(* POU LON/Module_1/Internal/FuSendCpValueReq_Module_1, ST *)
FUNCTION FuSendCpValueReq_Module_1 : BOOL
(******************************************)
(* Automatic generated code, do not edit! *)
(******************************************)
VAR_INPUT
	ptCp : POINTER TO BYTE;
	ptInternalUseOnly : POINTER TO BYTE;
	wCpIndex : WORD;
END_VAR
IF (ptCp <> 0) THEN
	IF ptInternalUseOnly^.0 = TRUE THEN
		OutDataTelegram_Module_1[0] := C2M_CP_VALUE_QRY;
		OutDataTelegram_Module_1[1] := WORD_TO_BYTE(wCpIndex AND 16#FF);
		OutDataTelegram_Module_1[2] := WORD_TO_BYTE((wCpIndex / 256) AND 16#FF);

		mbxModule_1.bTxPrio := 1;
		mbxModule_1.bTxProtID := 0;
		mbxModule_1.pbTxData := ADR(OutDataTelegram_Module_1);
		mbxModule_1.unTxLen := 3;
		mbxModule_1.MBX_SEND();

		IF (mbxModule_1.nError <> MBX_OK) THEN
			FuSendCpValueReq_Module_1 := FALSE;
			RETURN;
		END_IF
		ptInternalUseOnly^.0 := FALSE;
	END_IF
END_IF

FuSendCpValueReq_Module_1 := TRUE;
END_FUNCTION

(* POU LON/Shared/Internal/FuSnvtFilePosToRaw, ST *)
FUNCTION FuSnvtFilePosToRaw : BOOL
(******************************************)
(* Automatic generated code, do not edit! *)
(******************************************)
VAR_INPUT
	NvDataIn :  POINTER TO typSnvtFilePos;
	DataOut : POINTER TO ARRAY[0..5] OF BYTE;
END_VAR
VAR
END_VAR
DataOut^[0] := DINT_TO_BYTE(SHR(NvDataIn^.diRwPtr, 24));
DataOut^[1] := DINT_TO_BYTE(SHR(NvDataIn^.diRwPtr, 16));
DataOut^[2] := DINT_TO_BYTE(SHR(NvDataIn^.diRwPtr, 8));
DataOut^[3] := DINT_TO_BYTE(NvDataIn^.diRwPtr);

DataOut^[4] := WORD_TO_BYTE(SHR(NvDataIn^.wRwLength, 8));
DataOut^[5] := WORD_TO_BYTE(NvDataIn^.wRwLength);

FuSnvtFilePosToRaw := TRUE;
END_FUNCTION

(* POU LON/Shared/Internal/FuSnvtFileReqToRaw, ST *)
FUNCTION FuSnvtFileReqToRaw : BOOL
(******************************************)
(* Automatic generated code, do not edit! *)
(******************************************)
VAR_INPUT
	NvDataIn :  POINTER TO typSnvtFileReq;
	DataOut : POINTER TO ARRAY[0..11] OF BYTE;
END_VAR
VAR
END_VAR
DataOut^[0] := NvDataIn^.bRequest;

DataOut^[1] := WORD_TO_BYTE(SHR(NvDataIn^.wIndex, 8));
DataOut^[2] := WORD_TO_BYTE(NvDataIn^.wIndex);

DataOut^[3] := WORD_TO_BYTE(SHR(NvDataIn^.wReceiveTimeout, 8));
DataOut^[4] := WORD_TO_BYTE(NvDataIn^.wReceiveTimeout);

DataOut^[5] := NvDataIn^.abDestAddress[0];
DataOut^[6] := NvDataIn^.abDestAddress[1];
DataOut^[7] := NvDataIn^.abDestAddress[2];
DataOut^[8] := NvDataIn^.abDestAddress[3];
DataOut^[9] := NvDataIn^.abDestAddress[4];

DataOut^[10] := NvDataIn^.bAuthOn;

DataOut^[11] := NvDataIn^.bPrioOn;

FuSnvtFileReqToRaw := TRUE;
END_FUNCTION

(* POU LON/Shared/Internal/FuSnvtStateToRaw, ST *)
FUNCTION FuSnvtStateToRaw : BOOL
(******************************************)
(* Automatic generated code, do not edit! *)
(******************************************)
VAR_INPUT
	NvDataIn :  POINTER TO typSnvtState;
	DataOut : POINTER TO ARRAY[0..1] OF BYTE;
END_VAR
VAR
END_VAR
DataOut^[0] := NvDataIn^.bBitfieldByteOffset0;

DataOut^[1] := NvDataIn^.bBitfieldByteOffset1;

FuSnvtStateToRaw := TRUE;
END_FUNCTION

(* POU Utils Functions/LAMP_AL_GENERALE, ST *)
FUNCTION_BLOCK LAMP_AL_GENERALE
VAR_INPUT

	Allarme: BOOL;
	Warning: BOOL;
END_VAR
VAR_OUTPUT
	SistemaOK:BOOL;
	SistemaInAllarme:BOOL;
	SistemaWarning:BOOL;
	AllarmeLampada:BOOL;
END_VAR
VAR
	Lampeggio:BLINK;
END_VAR
IF Allarme THEN       					(* Se Allarme Attivo Lucde fissa ON *)
	SistemaInAllarme:=TRUE;
	SistemaWarning:=FALSE;
	AllarmeLampada:=TRUE;
ELSIF Warning THEN					(* Se Allarme Attivo Lucde fissa pulse *)
	SistemaInAllarme:=FALSE;
	SistemaWarning:=TRUE;
	Lampeggio(ENABLE:=TRUE , TIMELOW:=t#1s , TIMEHIGH:=t#1s , OUT=>AllarmeLampada );
ELSE
	SistemaInAllarme:=FALSE;
	SistemaWarning:=FALSE;
	AllarmeLampada:=FALSE;
END_IF
END_FUNCTION_BLOCK

(* POU Utils Functions/LINEAR, ST *)
FUNCTION LINEAR : REAL (* Linear interpolation *)
VAR_INPUT
	X_In	: REAL;
	P1_X	: REAL;
	P1_Y	: REAL;
	P2_X	: REAL;
	P2_Y	: REAL;
END_VAR
VAR
END_VAR
LINEAR:=P1_Y+(((P2_Y-P1_Y)*(X_In-P1_X))/(P2_X-P1_X));
END_FUNCTION

(* POU Utils Functions/LINEAR_BAD, ST *)
FUNCTION LINEAR_BAD : INT (* Linear interpolation *)
VAR_INPUT
	PuntoMinX	: INT;
	PuntoMaxX	: INT;
	ValIn		: INT;
	PuntoMinY	: REAL;
	PuntoMaxY	: REAL;
	Decimali	: BYTE;
END_VAR
VAR
	Gain				: REAL;
	PuntoMinX_R			: REAL;
	PuntoMaxX_R			: REAL;
	Linearizzazione_R	: REAL;
END_VAR
PuntoMinX_R:=INT_TO_REAL(PuntoMinX);
PuntoMaxX_R:=INT_TO_REAL(PuntoMaxX);

Gain:=(PuntoMaxX_R-PuntoMinX_R)/(PuntoMaxY-PuntoMinY);	(* Calcolo in guadagno per la linarizzazione *)
Linearizzazione_R:=PuntoMinx+(Gain*(ValIn-PuntoMinY));	(* Ottengo il valore linearizzato *)

LINEAR_BAD:=REAL_TO_INT(Linearizzazione_R*(EXPT(10, Decimali)));  (* Ottengo intero con i decimai voluti *)
END_FUNCTION

(* POU TCP_Logger/LogTrig, ST *)
FUNCTION LogTrig : BOOL
VAR
	s1 : STRING(160);
	i  : BYTE;
END_VAR
VAR_INPUT
END_VAR
(*---------------------------------------------------------------*)
	Logger_Head();
(*---------------------------------------------------------------*)

CTB01.AddLogData(MBUS:=MBUS01);

CTL01.AddLogData(COUNT:=Ctl01_Counter);
CTL02.AddLogData(COUNT:=Ctl02_Counter);

CAL01.AddLogData(CLIM:=CAL01_Clima);
CAL02.AddLogData(CLIM:=CAL02_Clima);

Logger.s1:='&PBV01=';
Logger.s1:=CONCAT(Logger.s1,SEL(ALARM_PB01,'1','0'));    (* 0= OK , 1 = Allarme *)
Logger.s1:=CONCAT(Logger.s1,';');
ADDSTRING(ADR(Logger.TData), ADR(Logger.s1), Logger.TLen);
Logger.s1:='&PBV02=';
Logger.s1:=CONCAT(Logger.s1,SEL(ALARM_PB02,'1','0'));    (* 0= OK , 1 = Allarme *)
ADDSTRING(ADR(Logger.TData), ADR(Logger.s1), Logger.TLen);


(* Modbus Pumps *)
CIR01.AddLogData(ModBus:=MODB01);
CIR02.AddLogData(ModBus:=MODB01);
CIR03.AddLogData();
CIRD01.AddLogData(ModBus:=MODB01);
CIRD02.AddLogData(ModBus:=MODB01);
CIRD03.AddLogData(ModBus:=MODB01);
CIRD04.AddLogData(ModBus:=MODB01);
CIRD05.AddLogData(ModBus:=MODB01);
CIRD06.AddLogData();

VRD01.AddLogData(CLIM:=VRD01_Clima);
VRD02.AddLogData(CLIM:=VRD02_Clima);
VRD03.AddLogData(CLIM:=VRD03_Clima);

TPV01.AddLogData();
TPV02.AddLogData();
TPV03.AddLogData();
TPV04.AddLogData();
TPV05.AddLogData();
TPV06.AddLogData();



ZTHL07.AddLogData(ModBus:=MODB02);
ZTHL08.AddLogData(ModBus:=MODB02);
ZTHL09.AddLogData(ModBus:=MODB02);
ZTHL10.AddLogData(ModBus:=MODB02);
ZTHL11.AddLogData(ModBus:=MODB02);
ZTHL12.AddLogData(ModBus:=MODB02);
ZTHL13.AddLogData(ModBus:=MODB02);

THER01.AddLogData();
THER02.AddLogData();
THER03.AddLogData();
THER04.AddLogData();
THER05.AddLogData();
THER06.AddLogData();
THER07.AddLogData();
THER250.AddLogData();

(*---------------------------------------------------------------*)
	Logger_Send();
(*---------------------------------------------------------------*)
END_FUNCTION

(* POU Utils Functions/MEAN_T, ST *)
FUNCTION MEAN_T : INT
VAR_INPUT
		T1		:	INT;
		T2		:	INT;

		THR_L	:	INT;
		THR_H	:	INT;
END_VAR
VAR
		Tmean	:	INT;
END_VAR
IF T1 >= THR_L AND T1 <= THR_H THEN

	IF T2 >= THR_L AND T2 <= THR_H THEN
		Tmean := (T1 + T2)/2;
	ELSE
		Tmean := T1;
	END_IF
ELSE
	IF T2 >= THR_L AND T2 <= THR_H THEN
		Tmean := T2;
	ELSE
		Tmean := 16#7FFF;	(* No valid temperature data has been passed *)
	END_IF
END_IF

MEAN_T := Tmean;
END_FUNCTION

(* POU Utils Functions/MEMCLR, ST *)
FUNCTION MEMCLR:BOOL
VAR_INPUT
	pDestinationAddress:POINTER TO ARRAY[1..2] OF BYTE;
	BytesToClear:WORD;
END_VAR
VAR
END_VAR
WHILE (BytesToClear > 0) DO
	pDestinationAddress^[1]:=0;
	pDestinationAddress:=ADR(pDestinationAddress^[2]); (* increment destination *)
	BytesToClear:=BytesToClear -1; (* decrement number of bytes to copy *)
END_WHILE
END_FUNCTION

(* POU LON/Module_1/ApplicationMessage/Module_1_ApplicationMsgSend, ST *)
FUNCTION_BLOCK Module_1_ApplicationMsgSend
(******************************************)
(* Automatic generated code, do not edit! *)
(******************************************)
VAR_INPUT
	xSend 		  : BOOL;
	abAddress     : ARRAY[0..10] OF BYTE;
	typServiceSend  : ServiceType;
	xPriority : BOOL;
	xAuthentification : BOOL;
	bMsgCodeSend  : BYTE;
	abMsgDataSend : ARRAY[0..47] OF BYTE;
	bLengthSend	  : BYTE;
END_VAR
VAR_OUTPUT
	bSendStatus   : BYTE;
END_VAR
VAR
	bAddressLength : BYTE;
	RtrigSend : R_TRIG;
END_VAR
RtrigSend(CLK:=xSend);
IF RtrigSend.Q AND (xInitRunning_Module_1 = FALSE) AND (mbxModule_1.bStatus.0) THEN
	OutDataTelegram_Module_1[0] := C2M_LON_MSG_SEND;
	OutDataTelegram_Module_1[1] := INT_TO_BYTE(typServiceSend);
	OutDataTelegram_Module_1[1].6 := xAuthentification;
	OutDataTelegram_Module_1[1].7 := xPriority;
	IF (abAddress[0] = 2) THEN
		bAddressLength := 11;
	ELSE
		bAddressLength := 5;
	END_IF
	FuMemCopy(ADR(abAddress), ADR(OutDataTelegram_Module_1[2]), bAddressLength);
	OutDataTelegram_Module_1[2+bAddressLength] := bMsgCodeSend;
	IF bLengthSend > 48 THEN bLengthSend := 48; END_IF;
	FuMemCopy(ADR(abMsgDataSend), ADR(OutDataTelegram_Module_1[2+bAddressLength+1]), bLengthSend);

	mbxModule_1.bTxPrio := BOOL_TO_BYTE(xPriority);
	mbxModule_1.bTxProtID := 0;
	mbxModule_1.pbTxData := ADR(OutDataTelegram_Module_1);
	mbxModule_1.unTxLen := 3 + bAddressLength + bLengthSend;
	mbxModule_1.MBX_SEND();

	IF (mbxModule_1.nError <> MBX_OK) THEN
		bSendStatus := 255;
	ELSE
		bSendStatus := 0;
	END_IF
END_IF
END_FUNCTION_BLOCK

(* POU LON/Module_1/ApplicationMessage/Module_1_ApplicationMsgSendRsp, ST *)
FUNCTION_BLOCK Module_1_ApplicationMsgSendRsp
(******************************************)
(* Automatic generated code, do not edit! *)
(******************************************)
VAR_INPUT
	xSend 	  : BOOL;
	bCorrelator : BYTE;
	bMsgCode  : BYTE;
	abMsgData : ARRAY[0..47] OF BYTE;
	bLength	  : BYTE;
END_VAR
VAR_OUTPUT
	bSendStatus : BYTE;
END_VAR
VAR
	RtrigSend : R_TRIG;
END_VAR
RtrigSend(CLK:=xSend);
IF RtrigSend.Q AND (xInitRunning_Module_1 = FALSE) AND (mbxModule_1.bStatus.0) THEN
	OutDataTelegram_Module_1[0] := C2M_LON_MSG_RSP_SEND;
	OutDataTelegram_Module_1[1] := bCorrelator;
	OutDataTelegram_Module_1[2] := bMsgCode;
	IF bLength > 48 THEN bLength := 48; END_IF;
	FuMemCopy(ADR(abMsgData), ADR(OutDataTelegram_Module_1[3]), bLength);

	mbxModule_1.bTxPrio := BOOL_TO_BYTE(bCorrelator.7);
	mbxModule_1.bTxProtID := 0;
	mbxModule_1.pbTxData := ADR(OutDataTelegram_Module_1);
	mbxModule_1.unTxLen := 3 + bLength;
	mbxModule_1.MBX_SEND();

	IF (mbxModule_1.nError <> MBX_OK) THEN
		bSendStatus := 255;
	ELSE
		bSendStatus := 0;
	END_IF
END_IF
END_FUNCTION_BLOCK

(* POU Utils Functions/MUX_T, ST *)
FUNCTION MUX_T : INT
(* Manage temperatures measured by different probes in the same room/environment, considering possible probe measurement errors *)
VAR_INPUT
	T1		:	INT;
	T2		:	INT;
	T3		:	INT;
	(*T4		:	INT := 0;*)

	Err1	:	BOOL := TRUE;
	Err2	:	BOOL := TRUE;
	Err3	:	BOOL := TRUE;
	(*Err4	:	BOOL := TRUE;*)

	Used	:	BYTE;

END_VAR
VAR
	Sum		:	INT;
	count	:	BYTE;
END_VAR
CASE Used OF

	1:	(* T1 passed *)
		IF Err1 THEN
			Sum := 16#7FFF;
		ELSE
			Sum := T1;
			count := 1;
		END_IF

	2:	(* T1, T2 passed *)
		IF Err1 THEN
			IF Err2 THEN
				Sum := 16#7FFF;
			ELSE
				Sum := T2;
				count := 1;
			END_IF
		ELSE
			IF Err2 THEN
				Sum := T1;
				count := 1;
			ELSE
				Sum := T1 + T2;
				count := 2;
			END_IF
		END_IF

	3:	(* T1, T2, T3 passed *)
		IF Err1 THEN
			IF Err2 THEN
				IF Err3 THEN
					Sum := 16#7FFF;
				ELSE
					Sum := T3;
					count := 1;
				END_IF
			ELSE
				IF Err3 THEN
					Sum := T2;
					count := 1;
				ELSE
					Sum := T2 + T3;
					count := 2;
				END_IF
			END_IF
		ELSE
			IF Err2 THEN
				IF Err3 THEN
					Sum := T1;
					count := 1;
				ELSE
					Sum := T1 + T3;
					count := 2;
				END_IF
			ELSE
				IF Err3 THEN
					Sum := T1 + T2;
					count := 2;
				ELSE
					Sum := T1 + T2 + T3;
					count := 3;
				END_IF
			END_IF
		END_IF
(*
	4:
		IF Err1 THEN
			IF Err2 THEN
				IF Err3 THEN
					IF Err4 THEN
						Sum := 16#7FFF;
					ELSE
						Sum := T4;
						count := 1;
					END_IF
				ELSE
					IF Err4 THEN
						Sum := T3;
						count := 1;
					ELSE
						Sum := T3 + T4;
						count := 2;
					END_IF
				END_IF
			ELSE
				IF Err3 THEN
					IF Err4 THEN
						Sum := T2;
						count := 1;
					ELSE
						Sum := T2 + T4;
						count := 2;
					END_IF
				ELSE
					IF Err4 THEN
						Sum := T2 + T3;
						count := 2;
					ELSE
						Sum := T2 + T3 + T4;
						count := 3;
					END_IF
				END_IF
			END_IF
		ELSE
			IF Err2 THEN
				IF Err3 THEN
					IF Err4 THEN
						Sum := T1;
					ELSE
						Sum := T1 + T4;
						count := 2;
					END_IF
				ELSE
					IF Err4 THEN
						Sum := T1 + T3;
						count := 2;
					ELSE
						Sum := T1 + T3 + T4;
						count := 3;
					END_IF
				END_IF
			ELSE
				IF Err3 THEN
					IF Err4 THEN
						Sum := T1 + T2;
						count := 2;
					ELSE
						Sum := T1 + T2 + T4;
						count := 3;
					END_IF
				ELSE
					IF Err4 THEN
						Sum := T1 + T2 + T3;
						count := 3;
					ELSE
						Sum := T1 + T2 + T3 + T4;
						count := 4;
					END_IF
				END_IF
			END_IF
		END_IF
*)
END_CASE

IF Sum = 16#7FFF THEN
	(* No valid data -> return default *)
	MUX_T := Plant_DefaultTAmb;
ELSE
	(* Do average *)
	MUX_T := Sum/count;
END_IF
END_FUNCTION

(* POU Plant_Objects/obj_CAL_VT100GC1B, ST *)
FUNCTION_BLOCK obj_CAL_VT100GC1B
(* === CALDAIA VIESSMAN via LON ===
   v1.0[16/04/15] - Versioning
*)
VAR_INPUT
	(* Settings *)
	ID				: BYTE;
	(* Controls *)
	Run				: BOOL;

	(* LON Status *)
	ModuleState	  : DWORD;
	(*** LON to CAL ***)
	(* Node inputs *)
	NO_Request    : typSnvtObjRequest;
	NO_TimeSet    : typSnvtTimeStamp;
	NO_AlarmSet   : typSnvtAlarm;
	(* Domestic hot water controller *)
	DHW_ModeSet   : typSnvtHvacMode;
	DHW_SetPoint  : typSnvtTempP;
	(* Central flow demand manager *)
	CFD_SetEnable : typSnvtSwitch;
	CFD_SetMode   : typSnvtHvacMode;
	CFD_SetPoint  : typSnvtTempP;
	(* LON From CAL *)
	NO_Status     : typSnvtObjStatus;
	NO_Alarm      : typSnvtAlarm;
	NO_RlyState   : typSnvtState;
	DHW_ActTemp   : typSnvtTempP;			(* Actual DHW temperature *)
	DHW_SetTemp   : typSnvtTempP;			(* Actual temperature set point *)
	CFD_GetEnable : typSnvtSwitch;
	CFD_Temp      : typSnvtTempP;
	CFD_SetTemp   : typSnvtTempP;


	(*Temperature	:	INT;*)

	SetPointManuale: INT; 			(* SetPoint forazato in manuale escludendo la curva di carico *)
	AbilitaSetPointManuale : BOOL ; (* Abilita il funzionamento col set point Manaule Escludendo la curva cliamtica *)


END_VAR
VAR_IN_OUT
	CLIM		  : typ_Clima;
END_VAR
VAR_OUTPUT
	Curve_Temp	: INT;

	(* Status *)
	Status_Log	: BYTE;
	Status_Vis 	: DWORD;
END_VAR
VAR
	InitOK		: BOOL;
	UpdateOK	: BOOL;
	fAlarm		: BOOL;
	fAlarmBUS	: BOOL;
	fWarning	: BOOL;

	Curve 		: CHARCURVE;
	Curve_Err 	: BYTE;

	Timer1		: TON  := ( PT:=T#5s);		(* Refresh timer for output vars *)

END_VAR
(* Check initialization *)
(*IF NOT InitOK THEN Init(); END_IF*)

(* Check LON connection *)
(*
...
*)

(* Check state *)
IF NO_Alarm.bAlarmType=1 THEN
	IF NOT fAlarm THEN
		fAlarm:=TRUE;
		LogEv(EL_Alarm,EO_CAL,ID,4,RAWTOHEXSTR(ADR(NO_Alarm.abAlarmLimit[2]),2));
	END_IF
ELSE
	IF fAlarm THEN
		LogEv(EL_LOg,EO_CAL,ID,6,'Allarme_Caldaia_Rientrato');
	END_IF
	fAlarm:=FALSE;
END_IF

(* Check climatic setup *)
IF NOT CLIM.InitOK THEN Clima_Default(); END_IF;
(* Calculate Setpoint *)
Curve(	IN:= T_AMB,	N:= 5, P:= CLIM.Points,
		OUT=> Curve_Temp, ERR=> Curve_Err );
IF Curve_Err>0 THEN
	IF NOT fWarning THEN
		fWarning:=TRUE;
		LogEv(EL_Wrn,EO_CAL,ID,2,'Climatic_Error');
	END_IF
ELSE
	fWarning:=FALSE;
END_IF

(* Scelta del set point della cladaia o vien preso dalla curva cliamtica o da un riferimento esterno *)
IF AbilitaSetPointManuale THEN
	CFD_SetPoint.iSnvtTempP:=(SetPointManuale+OffsetSetPointManuale)*10;
ELSE
	CFD_SetPoint.iSnvtTempP:=Curve_Temp*10;
END_IF

(* Attivazione caldaia *)
IF Run THEN
	CFD_SetMode.bSnvtHvacMode := 1;		(* Heat mode *)
ELSE
	CFD_SetMode.bSnvtHvacMode := 6;		(* Off *)
END_IF

(* Status color *)
   IF fAlarm OR fAlarmBUS	THEN Status_Log:=2; Status_Vis:=COLOR_RED;
ELSIF fWarning 		   		THEN Status_Log:=1; Status_Vis:=COLOR_YELLOW;
              				ELSE Status_Log:=0; Status_Vis:=SEL(Run,16#006000,16#20F020);
END_IF
END_FUNCTION_BLOCK
ACTION AddLogData:
Logger.s1:=INSERT('&CAL=',BYTE_TO_STRING(ID),4);
IF ID<10 THEN Logger.s1:=INSERT(Logger.s1,'0',4); END_IF

Logger.s1:=CONCAT(Logger.s1,INT_TO_STRING(CFD_SetPoint.iSnvtTempP/10));		Logger.s1:=CONCAT(Logger.s1,';');
Logger.s1:=CONCAT(Logger.s1,SEL(Run,'0','100'));							Logger.s1:=CONCAT(Logger.s1,';');

Logger.s1:=CONCAT(Logger.s1,WORD_TO_STRING(Status_Log));

Logger.s1:=CONCAT(Logger.s1,';');
Logger.s1:=CONCAT(Logger.s1,INT_TO_STRING(OffsetSetPointManuale));
Logger.s1:=CONCAT(Logger.s1,';');
Logger.s1:=CONCAT(Logger.s1,INT_TO_STRING(CFD_GetEnable.bValue/2)); (* Potenza Caldaia *)
Logger.s1:=CONCAT(Logger.s1,';');
Logger.s1:=CONCAT(Logger.s1,INT_TO_STRING(CFD_GetEnable.siState)); 	(* Presenza Fiamma *)
Logger.s1:=CONCAT(Logger.s1,';');
Logger.s1:=CONCAT(Logger.s1,INT_TO_STRING(CFD_Temp.iSnvtTempP/10)); 	(* Temp. Mandata da Caldaia*)

ADDSTRING(ADR(Logger.TData), ADR(Logger.s1), Logger.TLen);
END_ACTION
ACTION Clima_Default:
IF CLIM.Points[0].X=0 THEN
	CLIM.Points[0].X:=-300; CLIM.Points[0].Y:=770;
	CLIM.Points[1].X:=-70 ; CLIM.Points[1].Y:=770;
	CLIM.Points[2].X:= 80;  CLIM.Points[2].Y:=650;
	CLIM.Points[3].X:= 200; CLIM.Points[3].Y:=300;
	CLIM.Points[4].X:= 500; CLIM.Points[4].Y:=250;
END_IF
CLIM.InitOK:=TRUE;
LogEv(EL_Wrn,EO_CAL,ID,1,'Climatic_default');
END_ACTION
ACTION Heartbeat:
(* Call this at same cycle of LON execution call *)
Timer1(IN:=NOT Timer1.Q,PT:=T#1m);

NO_TimeSet.bDay := SYS.Time_Day;
NO_TimeSet.bMonth := SYS.Time_Month;
NO_TimeSet.iYear := SYS.Time_Year;
NO_TimeSet.bHour := SYS.Time_Hour;
NO_TimeSet.bMinute := SYS.Time_Minute;

NO_TimeSet.bStatusInformation:=SEL(Timer1.Q,0,16#80);
CFD_SetPoint.bStatusInformation:=SEL(Timer1.Q,0,16#80);		(* Re-trigger transmission every 60s *)
CFD_SetMode.bStatusInformation:=SEL(Timer1.Q,0,16#80);
(*CFD_SetEnable.bStatusInformation:=SEL(Timer1.Q,0,16#80);*)
END_ACTION
ACTION Init:
CFD_SetEnable.bValue:=0;

CFD_SetEnable.siState:=BYTE_TO_SINT(16#FF); (* Default value: AUTO *)

CFD_SetMode.bSnvtHvacMode:=16#FF; (* Default value: AUTO *)

(*CAL01.CFD_SetPoint.iSnvtTempP:=0; (* Default temperature: 0°C *)*)

(* End initialization *)
InitOK:=TRUE;
END_ACTION

(* POU Utils Functions/RAWTOHEXSTR, ST *)
FUNCTION RAWTOHEXSTR : STRING(128)
VAR_INPUT
	pData: POINTER TO BYTE;
	DataLen: BYTE;
END_VAR
VAR
	pt: POINTER TO BYTE;
	xl: BYTE;
END_VAR
pt:=ADR(RAWTOHEXSTR);

xl:=2;

WHILE DataLen>0 AND xl<128 DO

	pt^ := (pData^ / 16#10) + 48 + (((pData^ / 16#10)/10)*7);
	pt:=pt+1;
	pt^ := (pData^ AND 16#0F)  + 48 + (((pData^ AND 16#0F)/10)*7);
	pt:=pt+1;

	xl:=xl+2;

	DataLen:=DataLen-1;
	pData:=pData+1;

END_WHILE

pt^:=0;
END_FUNCTION

(* POU Plant_Objects/obj_CASCADE, ST *)
FUNCTION_BLOCK obj_CASCADE
VAR_INPUT
	RUN_Primary	:	BOOL;

	Tmonitor_On	:	TIME;	(* Wait time before enabling (switch on) second heater *)
	Tmonitor_Off:	TIME;	(* Wait time before disabling (switch off) second heater *)

	DeltaTempThr:	INT;	(* Delta temperature threshold at which enable monitoring *)

	SetTemp		:	INT;	(* Temperature setted *)
	ReadTemp	:	INT;	(* Temperature read on send way of heater *)

	TimerAttesaOn:TON;
	TimerAttesaOff:TOF;

END_VAR
VAR_OUTPUT
	OUT_Secondary	:	BOOL;	(* On/Off secondary heater *)
	State			:	BYTE;
END_VAR
VAR
	DeltaTemp	:	INT;
	Timer		:	TON;
END_VAR
DeltaTemp := SetTemp - ReadTemp;

(*

CASE State OF

	0:	(* Only primary heater works and delta temperature in the range *)
		IF RUN_Primary AND (DeltaTemp >= DeltaTempThr) THEN

				Timer.PT := Tmonitor_On;
				State := 1;

		END_IF

	1:	(* Only primary heater works and delta is out of the range -> Monitoring *)

		(* Used an hysteresys of 0.5°C	*)
		IF DeltaTemp >= (DeltaTempThr - 5) THEN

			Timer(IN:=NOT Timer.Q);

			IF Timer.Q THEN
				OUT_Secondary := TRUE;
				State := 2;

				Timer.PT := Tmonitor_Off;
				Timer(IN:=FALSE);
			END_IF
		ELSE
			Timer(IN:=FALSE);
			State := 0;
		END_IF

	2:	(* Both heaters working and monitoring delta for secondary heater off *)
		IF ReadTemp >= SetTemp THEN

			Timer(IN:=NOT Timer.Q);

			IF Timer.Q THEN
				OUT_Secondary := FALSE;
				State := 0;
				Timer(IN:=FALSE);
			END_IF

		ELSE
			Timer(IN:=FALSE);
		END_IF

END_CASE

*)
	IF RUN_Primary THEN

		TimerAttesaOn(IN:=(DeltaTemp >= DeltaTempThr) , PT:=Tmonitor_Off , Q=> , ET=> );
		TimerAttesaOff(IN:=TimerAttesaOn.Q, PT:=Tmonitor_On , Q=> , ET=> );
		OUT_Secondary:=TimerAttesaOff.Q;
	ELSE
		OUT_Secondary :=FALSE;
		TimerAttesaOn(IN:=FALSE , PT:=Tmonitor_Off , Q=> , ET=> );
		TimerAttesaOff(IN:=TimerAttesaOn.Q, PT:=t#1s , Q=> , ET=> );

	END_IF
END_FUNCTION_BLOCK

(* POU Plant_Objects/obj_CIR, ST *)
FUNCTION_BLOCK obj_CIR

(* === CIRCOLATORE STANDARD ===
   v1.0[16/04/15] - Versioning
   v1.1[11/08/15] - Added status reconstruction
*)
VAR CONSTANT
	SampleNr		: BYTE := 120;	(* 1 minute of observation *)
END_VAR
VAR_INPUT
	(* Settings *)
	ID				: BYTE;
	ExtStatus		: BOOL;	(* TRUE: external status signal input available, FALSE: no external status input *)

	(* Physical inputs (Force) *)
	CIR_RUN_REQ		: BOOL; (* External run request (no heat or cold requested) *)
	CIR_STOP_REQ	: BOOL; (* External stop request (has priority over RUN signals!) *)

	(* Physical inputs (Feedback) *)
	Pump_AL			: BOOL; (* Pump Alarm *)
	Pump_ST			: BOOL; (* Pump Status *)
	Pump_AUTO		: BOOL; (* Pump Auto/Manual *)

	(* Controls *)
	OnOff			: BOOL;	(* On/Off from chrono *)
	InitOK			: BOOL;

	(* Timings *)
	OnDelay		:	TIME;	(* Switch on delay *)
	OffDelay	:	TIME;	(* Switch off delay *)

	(* Input temperature needed if no real feedback about status is available *)
	Tprobe		:	INT;


END_VAR
VAR_OUTPUT
	CIR_EN			: BOOL;

	Ctrl_Run		: BOOL;		(* Logical status of the device: 0: Not running (switched off), 1: running *)
	Run				: BOOL;		(* Real status *)

	Status_Log		: WORD;
	Status_Vis		: DWORD;
END_VAR
VAR
	CIR_AUTO	: 	BOOL; (* Auto/Manual input signal *)
	Pump_En		:	BOOL;

	(* Filters *)
	fPump_ST	: 	FLT_TAP := (INITEV:=FALSE);
	fPump_En	:	FLT_EVENT;
	fCIR_AUTO	:	FLT_TAP;
	fStatus		:	FLT_EVENT;
	fStatusFault:	BOOL;

	(* Timer manage switch on/off delay *)
	Delay		: 	TONOF;

	(* Alarm and Warning counters *)
	AlarmCtr	:	BYTE;
	WarningCtr	:	BYTE;

	(* Filers on alarms and faults *)
	AlarmHw		:	FLT_TAP := (INITEV:=FALSE);

	(* Variables for status reconstruction *)
	aTprobe		:	ARRAY [1..SampleNr] OF INT;
	sample		:	BYTE;
	Tmean		:	INT;
	sum			:	INT;
	i			:	BYTE;
END_VAR
Init();

StatusRebuild();
(* Check alarms and warnings *)
CheckFault();

PumpManager();

IF AlarmCtr>0 THEN
	Status_Log := 2;
	Status_Vis := COLOR_RED;
ELSIF WarningCtr>0 OR fPump_ST.OUT THEN
	Status_Log := 1;
	Status_Vis := COLOR_YELLOW;
ELSE
	Status_Log := 0;
	Status_Vis := COLOR_GREEN;
END_IF
END_FUNCTION_BLOCK
ACTION AddLogData:
Logger.s1:=INSERT('&CIR=',BYTE_TO_STRING(ID),4);
IF ID<10 THEN Logger.s1:=INSERT(Logger.s1,'0',4); END_IF

Logger.s1:=CONCAT(Logger.s1,SEL(Pump_En,'0','100'));
Logger.s1:=CONCAT(Logger.s1,';');
Logger.s1:=CONCAT(Logger.s1,WORD_TO_STRING(Status_Log));
Logger.s1:=CONCAT(Logger.s1,';');
Logger.s1:=CONCAT(Logger.s1,SEL(CIR_RUN_REQ,'0','100'));
Logger.s1:=CONCAT(Logger.s1,';');
Logger.s1:=CONCAT(Logger.s1,SEL(CIR_STOP_REQ,'0','100'));


ADDSTRING(ADR(Logger.TData), ADR(Logger.s1), Logger.TLen);
END_ACTION
ACTION CheckFault:
(*** ALARMS ***)

(* Hardware alarm (physical input *)
AlarmHw(IN:=Pump_AL);

IF AlarmHw.EVH THEN
	LogEv(EL_Alarm,EO_CIR,ID,3,'');
	AlarmCtr := AlarmCtr + 1;
END_IF

IF AlarmHw.EVL THEN
	LogEv(EL_Log,EO_CIR,ID,4,'');
	AlarmCtr := SEL(AlarmCtr=0, AlarmCtr-1, 0);
END_IF

IF ExtStatus THEN
	fPump_ST(IN:=(Pump_ST<>CIR_EN));

	IF fPump_ST.EVH THEN
		IF Pump_AUTO THEN
			LogEv(SEL(Pump_ST,EL_Alarm,EL_Wrn),EO_CIR,ID,SEL(Pump_ST,5,6),'');
		ELSE
			LogEv(EL_Wrn,EO_CIR,ID,SEL(Pump_ST,1,2),'');
		END_IF
	END_IF

ELSE
	fPump_ST(IN:=fStatusFault);

	IF fPump_ST.EVH THEN
		IF Pump_AUTO THEN
			LogEv(SEL(OnOff,EL_Alarm,EL_Wrn),EO_CIR,ID,SEL(OnOff,5,6),'');
		ELSE
			LogEv(EL_Wrn,EO_CIR,ID,SEL(OnOff,1,2),'');
		END_IF
	END_IF
END_IF
END_ACTION
ACTION Init:
IF NOT InitOK THEN

	Delay.PT_OF := SEL(OffDelay=T#0ms, OffDelay, Plant_CirOffDelay);
	Delay.PT_ON := SEL(OnDelay=T#0ms, OnDelay, Plant_CirOnDelay) + WORD_TO_TIME(1000*ID);

	Pump_En := FALSE;

	InitOK := TRUE;

END_IF
END_ACTION
ACTION PumpManager:
(* Verify if in Auto or Manual mode *)
fCIR_AUTO(IN:=Pump_AUTO);

IF fCIR_AUTO.EVH THEN
	LogEv(EL_Log,EO_CIR,ID,8,'CIR_Auto');
	WarningCtr := SEL(WarningCtr=0, WarningCtr-1,0);
END_IF

(* Manual -> Keep switched on *)
IF fCIR_AUTO.EVL THEN
	LogEv(EL_Wrn,EO_CIR,ID,7,'CIR_Manual');
	WarningCtr := WarningCtr + 1;

	(* Switch on pump *)
	Pump_En := TRUE;
END_IF

(* Verify if OnOff is changed *)
Ctrl_Run := OnOff;

(* Check switch on or switch off delay *)
Delay(IN:=Ctrl_Run);

(* Do these instructions only if in AUTO mode *)
IF Pump_AUTO THEN
	(* If priority request *)
	IF CIR_STOP_REQ THEN Pump_En := FALSE;
	ELSIF CIR_RUN_REQ THEN Pump_En := TRUE;
	ELSE Pump_En := Delay.OUT;
	END_IF

	(* Set RUN signal (for external objects) *)
	IF AlarmHw.OUT THEN
		Run:=FALSE;
	ELSE
		Run:=Pump_En;
	END_IF
END_IF

(* Set value on physical outuput! *)
CIR_EN := Pump_En;
END_ACTION
ACTION StatusRebuild:
IF NOT ExtStatus THEN
	(* Check every 20 seconds *)
	IF  sample<sampleNr THEN
	
		aTprobe[sample] := Tprobe;
		sample := sample + 1;
	
	ELSE
	
		SHIFT_ARRAY(ADR(aTprobe),SampleNr);
	
		FOR i:=1 TO SampleNr BY 1 DO
			sum := sum + aTprobe[i];
		END_FOR
	
		Tmean := sum/SampleNr;
	
		(* CIR should be on but revealed temperature is decreasing *)
		IF OnOff AND (Tprobe<aTprobe[1]) THEN
			fStatusFault := TRUE;
		ELSE
			fStatusFault := FALSE;
		END_IF
	
		(* CIR should be off but revealed temperature is increasing *)
		IF NOT OnOff AND (Tprobe>aTprobe[1]) THEN
			fStatusFault := TRUE;
		ELSE
			fStatusFault := FALSE;
		END_IF
	END_IF
END_IF
END_ACTION

(* POU Utils Functions/TONOF, ST *)
FUNCTION_BLOCK TONOF
VAR_INPUT
	IN		: BOOL;
	PT_ON	: TIME; (* time to pass, before OUT is set *)
	PT_OF	: TIME; (* time to pass, before OUT is reset *)
END_VAR
VAR_OUTPUT
	OUT		: BOOL;
END_VAR
VAR
	timer	: TON;
END_VAR
IF IN<>OUT THEN
	timer(IN:=TRUE,PT:=SEL(IN,PT_OF,PT_ON));
	IF timer.Q THEN OUT:=IN; END_IF
ELSE
	timer(IN:=FALSE);
END_IF
END_FUNCTION_BLOCK

(* POU Plant_Objects/obj_CIR_DOPPIO_new, ST *)
FUNCTION_BLOCK obj_CIR_DOPPIO_new
(* === CIRCOLATORE GEMELLARE STANDARD ===
   v1.0[28/07/15] - Versioning
*)
VAR CONSTANT
	SampleNr		: BYTE := 120;	(* 1 minute of observation *)
END_VAR
VAR_INPUT
	(* Settings *)
	ID				: BYTE;
	ExtStatus		: BOOL;	(* TRUE: external status signal input available, FALSE: no external status input *)

	(* Physical inputs (Force) *)
	CIR_RUN_REQ		: BOOL; (* External run request (no heat or cold requested) *)
	CIR_STOP_REQ	: BOOL; (* External stop request (has priority over RUN signals!) *)

	(* Physical inputs (Feedback) *)
	PumpA_AL		: BOOL; (* Pump A Alarm *)
	PumpB_AL		: BOOL; (* Pump B Alarm *)
	PumpA_ST		: BOOL; (* Pump A Status *)
	PumpB_ST		: BOOL; (* Pump B Status *)
	PumpA_AUTO		: BOOL; (* Pump A Auto/Manual *)
	PumpB_AUTO		: BOOL; (* Pump B Auto/Manual *)

	(* Controls *)
	OnOff			: BOOL;	(* On/Off from chrono *)
	Mode			: BYTE;	(* Working mode: 0-Both pumps works simultaneously, 1-Alternate every 24h, 2-Master/Backup *)
	InitOK			: BOOL;

	(* Timings *)
	OnDelay		:	TIME;	(* Switch on delay *)
	OffDelay	:	TIME;	(* Switch off delay *)

	(* Input temperature needed if no real feedback about status is available *)
	Tprobe		:	INT;
END_VAR
VAR_OUTPUT
	PumpA_En		: BOOL;
	PumpB_En		: BOOL;

	Ctrl_Run		:	BOOL;		(* Logical status of the device: 0: Not running (switched off), 1: running *)
	Run				:	BOOL;		(* Real status *)

	Status_Log		: WORD;
	Status_Vis		: DWORD;
END_VAR
VAR
	CIR_AUTO	: BOOL; (* Auto/Manual input signal *)
	Pump_En		:	ARRAY [1..2] OF BOOL;

	ChangeTmr	: 	TON := (PT:=T#24h);			(* Timer that counts change time when in alternate mode *)
	ActivePump	: 	BYTE := 1;						(* Actual active pump *)
	NewActivePump	: BYTE := 1;

	(* Filters *)
	fPump_ST	: 	ARRAY [1..2] OF FLT_TAP := (INITEV:=FALSE);
	fPump_En	:	ARRAY [1..2] OF FLT_EVENT;
	fCIR_AUTO	:	ARRAY [1..2] OF FLT_TAP;
	fStatus		:	FLT_EVENT;
	fStatusFault:	BOOL;
	fBackup		:	FLT_EVENT := (INITEV:=FALSE);

	(* Timer manage switch on/off delay *)
	Delay		: 	TONOF;

	(* Alarm and Warning counters *)
	AlarmCtr	:	BYTE;
	WarningCtr	:	BYTE;

	(* Filers on alarms and faults *)
	AlarmHw		:	ARRAY [1..2] OF FLT_TAP := (INITEV:=FALSE);

	(* Variables for status reconstruction *)
	aTprobe		:	ARRAY [1..SampleNr] OF INT;
	sample		:	BYTE;
	Tmean		:	INT;
	sum			:	INT;
	i			:	BYTE;
END_VAR
Init();

PumpManager();

StatusRebuild();

(* Check alarms and warnings *)
CheckFault();

IF AlarmCtr>0 THEN
	Status_Log := 2;
	Status_Vis := COLOR_RED;
ELSIF WarningCtr>0 THEN
	Status_Log := 1;
	Status_Vis := COLOR_YELLOW;
ELSE
	Status_Log := 0;
	Status_Vis := COLOR_GREEN;
END_IF
END_FUNCTION_BLOCK
ACTION AddLogData:
Logger.s1:=INSERT('&CIRD=',BYTE_TO_STRING(ID),5);
IF ID<10 THEN Logger.s1:=INSERT(Logger.s1,'0',5); END_IF

Logger.s1:=CONCAT(Logger.s1,WORD_TO_STRING(Mode));			Logger.s1:=CONCAT(Logger.s1,';');

Logger.s1:=CONCAT(Logger.s1,SEL(Pump_En[1],'0','100'));		Logger.s1:=CONCAT(Logger.s1,';');
Logger.s1:=CONCAT(Logger.s1,SEL(Pump_En[2],'0','100'));		Logger.s1:=CONCAT(Logger.s1,';');

Logger.s1:=CONCAT(Logger.s1,WORD_TO_STRING(Status_Log));
Logger.s1:=CONCAT(Logger.s1,';');
Logger.s1:=CONCAT(Logger.s1,SEL(CIR_RUN_REQ,'0','100'));
Logger.s1:=CONCAT(Logger.s1,';');
Logger.s1:=CONCAT(Logger.s1,SEL(CIR_STOP_REQ,'0','100'));

ADDSTRING(ADR(Logger.TData), ADR(Logger.s1), Logger.TLen);
END_ACTION
ACTION CheckFault:
(*** ALARMS ***)

(**** PUMP 1 ****)

(* Hardware alarm (physical input *)
AlarmHw[1](IN:=PumpA_AL);

IF AlarmHw[1].EVH THEN
	LogEv(EL_Alarm,EO_CIRD,ID,3,'1');
	AlarmCtr := AlarmCtr + 1;
END_IF

IF AlarmHw[1].EVL THEN
	LogEv(EL_Log,EO_CIRD,ID,4,'1');
	AlarmCtr := SEL(AlarmCtr=0, AlarmCtr-1, 0);
END_IF

(**** PUMP 2 ****)

(* Hardware alarm (physical input *)
AlarmHw[2](IN:=PumpB_AL);

IF AlarmHw[2].EVH THEN
	LogEv(EL_Alarm,EO_CIRD,ID,3,'2');
	AlarmCtr := AlarmCtr + 1;
END_IF

IF AlarmHw[2].EVL THEN
	LogEv(EL_Log,EO_CIRD,ID,4,'2');
	AlarmCtr := SEL(AlarmCtr=0, AlarmCtr-1, 0);
END_IF



(* Check status *)
CASE Mode OF

	0:	(* Simultaneous *)

		IF ExtStatus THEN
			fPump_ST[1](IN:=(PumpA_ST<>PumpA_EN));

			IF fPump_ST[1].EVH THEN
				IF PumpA_AUTO THEN
					LogEv(SEL(PumpA_ST,EL_Alarm,EL_Wrn),EO_CIRD,ID,SEL(PumpA_ST,5,6),'1');
				ELSE
					LogEv(EL_Wrn,EO_CIRD,ID,SEL(PumpA_ST,1,2),'1');
				END_IF
			END_IF

			fPump_ST[2](IN:=(PumpB_ST<>PumpB_EN));

			IF fPump_ST[2].EVH THEN
				IF PumpB_AUTO THEN
					LogEv(SEL(PumpB_ST,EL_Alarm,EL_Wrn),EO_CIRD,ID,SEL(PumpB_ST,5,6),'2');
				ELSE
					LogEv(EL_Wrn,EO_CIRD,ID,SEL(PumpB_ST,1,2),'2');
				END_IF
			END_IF

		ELSE

			fPump_ST[1](IN:=fStatusFault);

			IF fPump_ST[1].EVH THEN
				IF PumpA_AUTO THEN
					LogEv(SEL(OnOff,EL_Alarm,EL_Wrn),EO_CIRD,ID,SEL(OnOff,5,6),'1');
					LogEv(SEL(OnOff,EL_Alarm,EL_Wrn),EO_CIRD,ID,SEL(OnOff,5,6),'2');
				ELSE
					LogEv(EL_Wrn,EO_CIRD,ID,SEL(OnOff,1,2),'1');
					LogEv(EL_Wrn,EO_CIRD,ID,SEL(OnOff,1,2),'2');
				END_IF
			END_IF

		END_IF

	1,2:	(*** Alternate working and Master/backup mode ***)

		IF ExtStatus THEN
			IF ActivePump=1 THEN

				fPump_ST[1](IN:=PumpA_ST<>PumpA_EN);

				IF fPump_ST[1].EVH THEN
					IF PumpA_AUTO THEN
						LogEv(SEL(PumpA_ST,EL_Alarm,EL_Wrn),EO_CIRD,ID,SEL(PumpA_ST,5,6),'1');
					ELSE
						LogEv(EL_Wrn,EO_CIRD,ID,SEL(PumpA_ST,1,2),'1');
					END_IF
				END_IF

			ELSE

				fPump_ST[2](IN:=PumpB_ST<>PumpB_EN);

				IF fPump_ST[2].EVH THEN
					IF PumpB_AUTO THEN
						LogEv(SEL(PumpB_ST,EL_Alarm,EL_Wrn),EO_CIRD,ID,SEL(PumpB_ST,5,6),'1');
					ELSE
						LogEv(EL_Wrn,EO_CIRD,ID,SEL(PumpB_ST,1,2),'2');
					END_IF
				END_IF
			END_IF

		ELSE

			fPump_ST[ActivePump](IN:=fStatusFault);

			IF fPump_ST[ActivePump].EVH THEN
				IF (PumpA_AUTO AND ActivePump=1) OR (PumpB_AUTO AND ActivePump=2) THEN

					LogEv(SEL(OnOff,EL_Alarm,EL_Wrn),EO_CIRD,ID,SEL(OnOff,5,6),BYTE_TO_STRING(ActivePump));

				ELSE

					LogEv(EL_Wrn,EO_CIRD,ID,SEL(OnOff,1,2),BYTE_TO_STRING(ActivePump));

				END_IF
			END_IF

		END_IF

END_CASE
END_ACTION
ACTION Init:
IF NOT InitOK THEN

	Delay.PT_OF := SEL(OffDelay=T#0ms, OffDelay, Plant_CirOffDelay);
	Delay.PT_ON := SEL(OnDelay=T#0ms, OnDelay, Plant_CirOnDelay) + WORD_TO_TIME(1000*ID);

	Pump_En[1] := FALSE;
	Pump_En[2] := FALSE;

	InitOK := TRUE;

END_IF
END_ACTION
ACTION PumpManager:
(* Verify if in Auto or Manual mode *)
fCIR_AUTO[1](IN:=PumpA_AUTO);
fCIR_AUTO[2](IN:=PumpB_AUTO);

(*** Pump A ***)
IF fCIR_AUTO[1].EVH THEN
	LogEv(EL_Log,EO_CIRD,ID,8,'1');
	WarningCtr := SEL(WarningCtr=0, WarningCtr-1,0);

	IF ActivePump=2 THEN Pump_En[1] := FALSE; END_IF
END_IF

(* Manual -> Keep switched on *)
IF fCIR_AUTO[1].EVL THEN
	LogEv(EL_Wrn,EO_CIRD,ID,7,'1');
	WarningCtr := WarningCtr + 1;

	(* Switch on pump A *)
	Pump_En[1] := TRUE;
END_IF

(*** Pump B ***)
IF fCIR_AUTO[2].EVH THEN
	LogEv(EL_Log,EO_CIRD,ID,8,'2');
	WarningCtr := SEL(WarningCtr=0, WarningCtr-1,0);

	IF ActivePump=1 THEN Pump_En[2] := FALSE; END_IF
END_IF

(* Manual -> Keep switched on *)
IF fCIR_AUTO[2].EVL THEN
	LogEv(EL_Wrn,EO_CIRD,ID,7,'2');
	WarningCtr := WarningCtr + 1;

	(* Switch on pump B *)
	Pump_En[2] := TRUE;
END_IF


(* Verify if OnOff is changed *)
Ctrl_Run := OnOff;

(* Check switch on or switch off delay *)
Delay(IN:=Ctrl_Run);

(* If working mode is Alternate, count change time *)
IF Mode=1 THEN

	ChangeTmr(IN:=NOT ChangeTmr.Q);

	IF ChangeTmr.Q THEN

		NewActivePump := SEL(ActivePump=1,1,2);
	
		(* If no alarm on other pump, keep going with the switch *)
		IF NOT AlarmHw[NewActivePump].OUT THEN	ActivePump := NewActivePump;
		ELSE LogEv(EL_Wrn,EO_CIRD,ID,15,'');		(* Pump not switched because of other pump's failure *)
		END_IF
	
		(* Switch off old active pump *)
		IF ActivePump=1 THEN Pump_En[2] := FALSE;
		ELSE Pump_En[1] := FALSE;
		END_IF
	
		ChangeTmr.PT := T#24h;
	END_IF
END_IF


(* Set output according to actual function mode *)
CASE Mode OF

	0:	(*** Simultaneous pumps working ***)
		IF PumpA_AUTO THEN

			IF CIR_STOP_REQ THEN Pump_En[1] := FALSE;
			ELSIF CIR_RUN_REQ THEN Pump_En[1] := TRUE;
			ELSE Pump_En[1] := Delay.OUT;
			END_IF

			(* Set RUN signal (for external objects) *)
			IF AlarmCtr>0 THEN (*OR fPump_ST[1].OUT OR fPump_ST[2].OUT THEN*)
				Run:=FALSE;
			ELSE
				Run:=Pump_En[1];
			END_IF
		END_IF

		IF PumpB_AUTO THEN

			IF CIR_STOP_REQ THEN Pump_En[2] := FALSE;
			ELSIF CIR_RUN_REQ THEN Pump_En[2] := TRUE;
			ELSE Pump_En[2] := Delay.OUT;
			END_IF

			(* Set RUN signal (for external objects) *)
			IF AlarmCtr>0 THEN (*OR fPump_ST[1].OUT OR fPump_ST[2].OUT THEN*)
				Run:=FALSE;
			ELSE
				Run:=Pump_En[2];
			END_IF
		END_IF

	1,2:  (*** Alternate working and Master/backup mode ***)
		IF fCIR_AUTO[ActivePump].OUT THEN

			(* If priority request *)
			IF CIR_STOP_REQ THEN Pump_En[ActivePump] := FALSE;
			ELSIF CIR_RUN_REQ THEN Pump_En[ActivePump] := TRUE;
			ELSE Pump_En[ActivePump] := Delay.OUT;
			END_IF

			fBackup(IN:=AlarmHw[ActivePump].OUT);

			IF fBackup.EVH THEN
				(* Pump switched because of current pump failure *)
				ActivePump := SEL(ActivePump=1,1,2);
				LogEv(EL_Wrn,EO_CIRD,ID,16,'');

				(* Switch off old active pump *)
				IF ActivePump=1 THEN Pump_En[2] := FALSE;
				ELSE Pump_En[1] := FALSE;
				END_IF
			END_IF


			(* Set RUN signal (for external objects) *)
			IF AlarmHw[1].OUT AND AlarmHw[2].OUT THEN
				Run:=FALSE;
			ELSE
				Run:=Pump_En[ActivePump];
			END_IF

		END_IF

END_CASE

(* Set value on physical outuput! *)
PumpA_En := Pump_En[1];
PumpB_En := Pump_En[2];
END_ACTION
ACTION StatusRebuild:
(* Check every 20 seconds *)
IF  sample<sampleNr THEN

	aTprobe[sample] := Tprobe;
	sample := sample + 1;

ELSE

	SHIFT_ARRAY(ADR(aTprobe),SampleNr);

	FOR i:=1 TO SampleNr BY 1 DO
		sum := sum + aTprobe[i];
	END_FOR

	Tmean := sum/SampleNr;

	(* CIR should be on but revealed temperature is decreasing *)
	IF OnOff AND (Tprobe<aTprobe[1]) THEN
		fStatusFault := TRUE;
	ELSE
		fStatusFault := FALSE;
	END_IF

	(* CIR should be off but revealed temperature is increasing *)
	IF NOT OnOff AND (Tprobe>aTprobe[1]) THEN
		fStatusFault := TRUE;
	ELSE
		fStatusFault := FALSE;
	END_IF
END_IF
END_ACTION

(* POU Plant_Objects/obj_CRON_EDITOR_01, ST *)
FUNCTION_BLOCK obj_CRON_EDITOR_01
(* === EDITOR CRONOGRAFO ===
   v1.0[16/04/15] - Versioning
   v1.1[19/05/15] - Create empty profile when not found
*)
VAR_INPUT

	(* Common selections *)
	CN_Sel:			BYTE:=1;
	CN_Act:			BYTE;
	CN_YSel:		WORD:=2015;
	CN_YAct:		WORD;

	(* Profile editor *)
	PR_Sel: 		BYTE:=1;
	PR_Act:			BYTE;
	PR_TT:			REAL;
	PR:				typ_Cron_Profile;
	(* Profile signals *)
	PR_Load:		BOOL;
	PR_Save:		BOOL;

	(* Calendar editor *)
	CA_Sel:			BYTE:=1; (* Calendar month selected *)
	CA_Act:			BYTE;    (* Calendar month active *)
	CA_DayF:		BYTE:=0;
	CA_DayL:		BYTE:=31;
	CA_TPR:			BYTE;
	CA:				typ_Cron_Calendar; (* Only used for first 32 entries *)
	(* Calendar signals *)
	CA_Load:		BOOL;
	CA_Save:		BOOL;

	(* Jolly editor *)
	JL:				ARRAY[0..9] OF typ_Cron_Jolly;
	(* Jolly signals *)
	JL_Load:		BOOL;
	JL_Save:		BOOL;

END_VAR
VAR_OUTPUT
	Message		: STRING;
END_VAR
VAR
	sFileName	: STRING;
	sFileMode	: STRING;
	hFile		: DWORD;
	Buf			: ARRAY[0..512] OF BYTE; (* AVOID THIS!! *)

	i			: WORD;
	ver			: BYTE;
	r1			: BOOL;
	r2			: DWORD;

	x: INT;
	maxProfili: INT;

	sFileNameOld	: STRING;
	sFileModeOld		: STRING;
	hFileOld			: DWORD;




	strAppoggio: STRING;
	FileGiaCreato: BOOL;
	fileCopiato: UDINT;

	tempMultiAnnoMax:INT;
	tempMultiAnnoIndex:INT;
	TEMP_MULTIANNO_MAX_DELTA:INT:=5;
	tempRicercaFileAnno:INT;
	tempAnno:INT;
	tempTrovato:BOOL;
END_VAR
IF PR_Load THEN PR_Load_Exe();
	PR_Load:=FALSE;
END_IF
IF PR_Save THEN
PR_Save_Exe();
PR_Save:=FALSE;
END_IF
IF CA_Load THEN
CA_Load_Exe();
CA_Load:=FALSE;
END_IF
IF CA_Save THEN
CA_Save_Exe();
CA_Save:=FALSE;
END_IF
IF JL_Load THEN
JL_Load_Exe();
JL_Load:=FALSE;
END_IF
IF JL_Save THEN
 JL_Save_Exe();
 JL_Save:=FALSE;
 END_IF
END_FUNCTION_BLOCK
ACTION CA_Load_Exe:
sFileMode:='r';
FileOpen();

IF hFile<>0 THEN

	(* Read calendar month *)
	FOR i := 0 TO 31 DO
		r1:=SysFileSetPos(File:=hFile, Pos:=(1024 + ((CA_Sel-1)*32 + i)*4));
		r2:=SysFileRead(File:=hFile, Buffer:=ADR(CA.Profile[i]), Size:=1);
	END_FOR

	(* Close file *)
	SysFileClose(File:=hFile);

	(* Validate data *)
	CA_Act :=CA_Sel;
	CN_Act :=CN_Sel;
	CN_YAct:=CN_YSel;

	Message:='Calendar load OK';

END_IF
END_ACTION
ACTION CA_Save_Exe:
sFileMode:='a';
FileOpen();

IF hFile<>0 THEN

	(* Write calendar month *)
	FOR i := 0 TO 31 DO
		r1:=SysFileSetPos(File:=hFile, Pos:=(1024 + ((CA_Sel-1)*32 + i)*4));
		r2:=SysFileGetPos(hFile);
		r2:=SysFileWrite(File:=hFile, Buffer:=ADR(CA.Profile[i]), Size:=1);
	END_FOR

	(* Close file *)
	SysFileClose(File:=hFile);

	Message:='Calendar save OK';

	(* db commentato! non salva i profili, ma solo il profilo corrente, che può anche essere modificato!*)
          (*PR_Save_exe();*)
	(* nel salvare il calendario aggiorno anche i profili così ho il file completo dei profili *)


END_IF

IF hFile<>0 THEN SysFileClose(File:=hFile); END_IF (*diego add*)
END_ACTION
ACTION FileOpen:
(* Create current filename 'yyyyCRnn.DAT' *) (* creo il nome del file da aparire *)
sFileName:=CONCAT(FilesPath,WORD_TO_STRING(CN_YSel));
sFileName:=CONCAT(STR1:=sFileName, STR2:='CR');
IF CN_Sel<10 THEN
sFileName:=CONCAT(STR1:=sFileName, STR2:='0');
END_IF
sFileName:=CONCAT(STR1:=sFileName, STR2:=BYTE_TO_STRING(CN_Sel));
sFileName:=CONCAT(STR1:=sFileName, STR2:='.DAT');


(* Apro il fiel in lettura per verificare se è presente altrimenti devo crearne uno nuovo a duplicare quello dell'anno precedente - apro 1  *)
hFile:=SysFileOpen(FileName:=sFileName, Mode:='r');
FileGiaCreato:=FALSE;

tempAnno:=CN_YSel;
tempTrovato:=FALSE;

(* File non trovato da creare  *)
IF hFile=0 THEN

	 (*cerco i file precendti: dall'anno prima fino a - TEMP_MULTIANNO_MAX_DELTA*)
	 tempRicercaFileAnno:=1;

	WHILE tempRicercaFileAnno<=TEMP_MULTIANNO_MAX_DELTA AND NOT tempTrovato DO


		strAppoggio:=INT_TO_STRING(tempAnno);
		(* Verifico se esite un file da cui partire *)
		StrAppoggio:=WORD_TO_STRING(STRING_TO_WORD(strAppoggio)-tempRicercaFileAnno);
		sFileNameOld:=CONCAT(FilesPath,StrAppoggio);

		sFileNameOld:=CONCAT(STR1:=sFileNameOld, STR2:='CR');
		IF CN_Sel<10 THEN
			sFileNameOld:=CONCAT(STR1:=sFileNameOld, STR2:='0');
		END_IF
		sFileNameOld:=CONCAT(STR1:=sFileNameOld, STR2:=BYTE_TO_STRING(CN_Sel));
		sFileNameOld:=CONCAT(STR1:=sFileNameOld, STR2:='.DAT');

		(* Apro il file in lettura per la verifica della presenza del file da copiare  *)
		hFileold:=SysFileOpen(FileName:=sFileNameOld, Mode:='r');

		IF hFileold<>0 THEN

			tempTrovato:=TRUE;

			fileCopiato:=SysFileCopy(sFileName,sFileNameold);

    		   	FileGiaCreato:=fileCopiato<>0;

			IF FileGiaCreato THEN
				Message:='File Sorgente/copia  trovato - file Copiato';
			ELSE
				Message:='File Sorgente/copia  trovato - file NON Copiato';
			END_IF


			(* Chiudo il file aperto per la verifica del file presente *)
			SysFileClose(File:=hFile);
			(* Chiudo il file aperto in lettura per la verifica della presenza del file da copiare  *)
			SysFileClose(File:=hFileold);

		END_IF

		tempRicercaFileAnno:=tempRicercaFileAnno+1;

	END_WHILE

	(* se non ho trovato nessun file..lo creo vuoto*)
	IF tempTrovato=FALSE THEN   (* file non trovato quindi devo crearne uno nuovo *)

			(* Create empty file *)
			hFile:=SysFileOpen(FileName:=sFileName, Mode:='w');
			MEMCLR(pDestinationAddress:=ADR(Buf), BytesToClear:=SIZEOF(Buf));
			FOR i := 0 TO 10239 BY 512 DO
				SysFileWrite(File:=hFile, Buffer:=ADR(Buf), Size:=512);
			END_FOR

			Buf[0]:=1;
			SysFileSetPos(File:=hFile, Pos:=0);
			SysFileWrite(File:=hFile, Buffer:=ADR(Buf), Size:=1);

			(* Chiudo il file aperto per la verifica del file presente *)
			SysFileClose(File:=hFile);
			(* Chiudo il file aperto in lettura per la verifica della presenza del file da copiare  *)
			SysFileClose(File:=hFileold);

			Message:='File Sorgente/copia non trovato-file Vuoto';

	END_IF


ELSE

	(* Chiudo il file aperto per la verifica del file presente *)
	SysFileClose(File:=hFile);

END_IF




(* Apro il file per permettere la scrittura o la lettura del file da parte delle altre action . la chiusura del file è delegata alle Action *)
hFile:=SysFileOpen(FileName:=sFileName, Mode:=sFileMode);
END_ACTION
ACTION JL_Load_Exe:
sFileMode:='r';
FileOpen();

IF hFile<>0 THEN

	(* Read jolly *)
	r1:=SysFileSetPos(File:=hFile, Pos:=512);
	r2:=SysFileRead(File:=hFile, Buffer:=ADR(JL), Size:=SIZEOF(JL));

	(* Close file *)
	SysFileClose(File:=hFile);

	(* Validate data *)
	CN_Act:=CN_Sel;
	CN_YAct:=CN_YSel;

	Message:='Jolly load OK';

END_IF
END_ACTION
ACTION JL_Save_Exe:
sFileMode:='a';
FileOpen();

IF hFile<>0 THEN

	(* Write selected profile *)
	r1:=SysFileSetPos(File:=hFile, Pos:=512);
	r2:=SysFileWrite(File:=hFile, Buffer:=ADR(JL), Size:=SIZEOF(JL));

	(* Close file *)
	SysFileClose(File:=hFile);

	Message:='Jolly save OK';

END_IF
END_ACTION
ACTION PR_Load_Exe:
sFileMode:='r';
FileOpen();

IF hFile<>0 THEN

	(* Read selected profile *)
	r1:=SysFileSetPos(File:=hFile, Pos:=(3072 + 512*PR_Sel));
	r2:=SysFileRead(File:=hFile, Buffer:=ADR(PR), Size:=SIZEOF(PR));

	(* Close file *)
	SysFileClose(File:=hFile);

	(* Validate data *)
	PR_Act:=PR_Sel;
	CN_Act:=CN_Sel;
	CN_YAct:=CN_YSel;

	Message:='Profile load OK';

END_IF
END_ACTION
ACTION PR_Save_Exe:
sFileMode:='a';
FileOpen();

IF hFile<>0 THEN

		(* Write selected profile *)
		r1:=SysFileSetPos(File:=hFile, Pos:=(3072 + 512*PR_Sel));
		r2:=SysFileWrite(File:=hFile, Buffer:=ADR(PR), Size:=SIZEOF(PR));

		(* Close file *)
		SysFileClose(File:=hFile);

		Message:='Profile save OK';

END_IF

IF hFile<>0 THEN SysFileClose(File:=hFile); END_IF (*diego add*)
END_ACTION
ACTION PR_Save_Exe_Multi:
(*eseguo  salvataggio profilo per l'anno corrente del CronoEditor - quello indicato da CN_YSel*)
CronEd.PR_Save_Exe();

(*verifico se esistono i file di schedulazioni per anni successivi: se aggiorno i profili anche lì*)

(*tempMultiAnnoMax dice fino a quale anno si considera*)
tempMultiAnnoMax:=CronEd.CN_YSel+TEMP_MULTIANNO_MAX_DELTA;

(* per ogni anno, vrifico se esiste il relativo file e se si aggiorno i profili anche li *)
FOR tempMultiAnnoIndex:=CronEd.CN_YSel+1 TO tempMultiAnnoMax BY 1 DO

	sFileName:=CONCAT(FilesPath,INT_TO_STRING(tempMultiAnnoIndex));
	sFileName:=CONCAT(STR1:=sFileName, STR2:='CR');
	IF CN_Sel<10 THEN
		sFileName:=CONCAT(STR1:=sFileName, STR2:='0');
	END_IF
	sFileName:=CONCAT(STR1:=sFileName, STR2:=INT_TO_STRING(CN_Sel));
	sFileName:=CONCAT(STR1:=sFileName, STR2:='.DAT');

	hFile:=SysFileOpen(FileName:=sFileName, Mode:='r');
	(* file esiste, aggiorno profili per quell'anno *)
	IF hFile<>0 THEN

		SysFileClose(File:=hFile);
		CronEd.CN_YSel:=tempMultiAnnoIndex;
		CronEd.PR_Save_Exe();

	ELSE
		SysFileClose(File:=hFile);

	END_IF


END_FOR
END_ACTION

(* POU Plant_Objects/obj_CRONTER_01, ST *)
FUNCTION_BLOCK obj_CRONTER_01
(* === THERMOSTAT ===
   v1.0[30/07/15] - Versioning
*)
VAR_INPUT
	(* Settings *)
	ID			: BYTE;		(* Index of instanced object *)

	InitOK		: BOOL;
	Alarm		: BOOL;
	Warning		: BOOL;

	Profile		: typ_Cron_Profile; 				(* Profilo attivo *)
	ProfileNr	: BYTE;								(* Indice profilo attivo *)
	CalendarIdx : WORD;								(* Indice calendario attivo *)
	Jolly		: ARRAY[0..9] OF typ_Cron_Jolly;	(* Jolly attivi *)

	Temperature	: INT;
	Local_MaxRunTAmb	:	INT;					(* Local maximum environment temperature, NOT "TAMB" *)
	Histeresys:INT; (* isteresi per la ripartenza del Comando ON*)


	sFile: 	STRING;


END_VAR
VAR_IN_OUT
END_VAR
VAR_OUTPUT
	SetPoint		: INT;
	Run				: BOOL;
	AntifreezeForce	: BOOL;
	RunCrono		: BOOL;

	(* Status *)
	Status_Log		: BYTE;
	Status_Vis 		: DWORD;
END_VAR
VAR
	Buf: 	ARRAY[0..512] OF BYTE; (* AVOID THIS!! *)
	hFile: 	DWORD;

	sFile2: STRING;

	i:		WORD;
	t1:		DWORD;
	t2:		BOOL;

END_VAR
(* Check initialization *)
(*IF NOT InitOK THEN Init(); END_IF*)

(* Check Temperature *)
IF Temperature <Local_MaxRunTAmb THEN

	(* LOCAL environment temperature lower than maximum allowed -> Proceed with SetPoint adjustment *)
	(* Chrono *)
(*	IF CalendarIdx<>Sys.Time_CT_Day THEN DB_Load(); END_IF *)

	IF CalendarIdx<>Sys.Time_CT_Day OR InitOK=FALSE THEN  (* col cambio della data carico il file corretti dove è intergrato il controllo della presenza del file *)
		CronEd(CN_Sel:=WORD_TO_BYTE(id),CN_YSel:=Sys.Time_Year, CA_Load:=TRUE,PR_Load:=TRUE);
		DB_Load(	sFile:= CronEd.sFileName);  (* aggiorno il SetPoint  partendo dal file noto*)
		InitOK:=TRUE;
	END_IF


	SetPoint:=Profile.Setpoint[Sys.Time_CT_Quarter];

	(* Check jolly *)
	FOR i := 0 TO 9 DO
		IF ( DT_TO_DWORD(Jolly[i].Start)>0  AND Jolly[i].End>Jolly[i].Start AND
		     Jolly[i].Start<=Sys.Time_CT_DT AND Jolly[i].End>Sys.Time_CT_DT ) THEN
				SetPoint:=Jolly[i].Temp;
		END_IF
	END_FOR

(*
	IF SetPoint < 180 THEN
		(* Switch off the device *)
		Run := FALSE;
	ELSE
		(* Set according to feedback T - Histeresys of 1°C *)
		IF Temperature >= (SetPoint + 5) THEN
			Run := FALSE;
		ELSIF Temperature <= (SetPoint - 5) THEN
			Run := TRUE;
		END_IF

		(* Between "SetPoint-5" and "SetPoint+5" last state (ON or OFF) of "Run" is kept	*)
	END_IF
*)
(* Gestione uscita Crono *)
		IF SetPoint>0 THEN RunCrono := TRUE;
		ELSIF SetPoint=0 THEN RunCrono := FALSE;
		END_IF

(* GEstione uscita Cronotermostato *)

		IF Temperature >= (SetPoint) THEN
			Run := FALSE;
		ELSIF Temperature <= (SetPoint - Histeresys) THEN
			Run := TRUE;
		END_IF
ELSE
	(* Environment overtemperature: stop heating -> Stop device *)
	Run := FALSE;
END_IF

(* Freeze warning: Switch on and heat! *)
(*IF Temperature < Plant_AntiFreezeTAmb THEN AntifreezeForce := TRUE;
ELSE AntifreezeForce := FALSE;
END_IF*)



(* Status color *)
   IF Alarm   THEN Status_Log:=2; Status_Vis:=COLOR_RED;
ELSIF Warning THEN Status_Log:=1; Status_Vis:=COLOR_YELLOW;
              ELSE Status_Log:=0; Status_Vis:=COLOR_GREEN;
			  END_IF
END_FUNCTION_BLOCK
ACTION AddLogData:
Logger.s1:=INSERT('&THER=',BYTE_TO_STRING(ID),5);
IF ID<10 THEN Logger.s1:=INSERT(Logger.s1,'0',5); END_IF

Logger.s1:=CONCAT(Logger.s1,INT_TO_STRING(SetPoint));			Logger.s1:=CONCAT(Logger.s1,';');

Logger.s1:=CONCAT(Logger.s1,WORD_TO_STRING(Status_Log));
ADDSTRING(ADR(Logger.TData), ADR(Logger.s1), Logger.TLen);
END_ACTION
ACTION DB_Create:
(* Create empty file *)
hFile:=SysFileOpen(FileName:=sFile, Mode:='w');

MEMCLR(pDestinationAddress:=ADR(Buf), BytesToClear:=SIZEOF(Buf));
FOR i := 0 TO 10239 BY 512 DO
	t1:=SysFileWrite(File:=hFile, Buffer:=ADR(Buf), Size:=512);		(* Clear created file (all bytes 0) *)
END_FOR
Buf[0]:=1;
t2:=SysFileSetPos(File:=hFile, Pos:=0);
t1:=SysFileWrite(File:=hFile, Buffer:=ADR(Buf), Size:=1);
SysFileClose(File:=hFile);
END_ACTION
ACTION DB_Load:
(*

DB_SetName();


(* File not found *)
IF hFile=0 THEN
	Warning:=TRUE;
	LogEv(EL_Wrn,EO_CRON,ID,1,'No_data_file');
	DB_Create();
	(* Reopen file *)
	hFile:=SysFileOpen(FileName:=sFile, Mode:='r');
	IF hfile=0 THEN
		Alarm:=TRUE;
		LogEv(EL_Alarm,EO_CRON,ID,3,'Filesystem_error');
		RETURN;
	END_IF
END_IF
*)

(* Open data file *)
hFile:=SysFileOpen(FileName:=sFile, Mode:='r');

(* Check version *)
SysFileRead(File:=hFile, Buffer:=ADR(Buf), Size:=1);
IF Buf[0]<>1 THEN
	IF NOT Alarm THEN
		Alarm:=TRUE;
		LogEv(EL_Alarm,EO_CRON,ID,2,'Bad_data_version');
	END_IF
	SysFileClose(File:=hFile);
	RETURN;
END_IF

(* Read Jolly data *)
t2:=SysFileSetPos(File:=hFile, Pos:=512);
t1:=SysFileRead(File:=hFile, Buffer:=ADR(Jolly), Size:=SIZEOF(Jolly));
(* Read active profile index *)
CalendarIdx:=Sys.Time_CT_Day;
t2:=SysFileSetPos(File:=hFile, Pos:=(1024+4*CalendarIdx));
t1:=SysFileRead(File:=hFile, Buffer:=ADR(ProfileNr), Size:=SIZEOF(ProfileNr));
(* Read active profile *)
t2:=SysFileSetPos(File:=hFile, Pos:=(3072+512*ProfileNr));
t1:=SysFileRead(File:=hFile, Buffer:=ADR(Profile), Size:=SIZEOF(Profile));

(* Close file and validate data *)
SysFileClose(File:=hFile);
END_ACTION
ACTION DB_SetName:
(* Create current filename 'yyyyCRnn.DAT' *)
sFile:=CONCAT(FilesPath,WORD_TO_STRING(Sys.Time_Year));
sFile:=CONCAT(STR1:=sFile, STR2:='CR');
IF ID<10 THEN
sFile:=CONCAT(STR1:=sFile, STR2:='0');
END_IF
sFile:=CONCAT(STR1:=sFile, STR2:=BYTE_TO_STRING(ID));
sFile:=CONCAT(STR1:=sFile, STR2:='.DAT');
END_ACTION
ACTION Init:
DB_Load();
InitOK:=TRUE;
END_ACTION

(* POU Plant_Objects/obj_CTL, ST *)
FUNCTION_BLOCK obj_CTL
(* === PULSE VOLUME COUNTER ===
   v1.0[16/04/15] - Versioning
*)
VAR_INPUT
	(* Settings *)
	ID				: BYTE;	(* Index of instanced object *)
	Peso			: DWORD;
	(* Physical inputs *)
	CTL_ST			: BOOL;
END_VAR
VAR_IN_OUT
	COUNT			: DWORD;
END_VAR
VAR_OUTPUT
	(* Status *)
	Status_Log		: BYTE;
END_VAR
VAR
	Filter			: FLT_TAP := ( INITEV:=FALSE );
	Timer			: TON;
	TCount			: DWORD;
	i				: DWORD;
END_VAR
(* Execute timer *)
Timer(IN:=NOT Timer.Q, PT:=T#60m);

(* Execute filter on counter status *)
Filter(IN:=CTL_ST);

(* Count event *)
IF Filter.EVH THEN
	COUNT:=COUNT+Peso;
	TCount:=TCount+1;
	(* Check flow rate *)
	IF TCount>=Plant_MaxWaterLoss THEN
		i:=(TCount*TIME_TO_DWORD(Timer.PT))/TIME_TO_DWORD(Timer.ET);	(* Estimated mc per hour *)
		i:= i * Peso;

		(* NB The weight is multiplied by 10 -> Need to divide it by 10 server side *)
		LogEv(EL_AlarmStop,EO_CTL,ID,1,DWORD_TO_STRING(i));
		Status_Log:=2;

		TCount:=0;
		Timer(IN:=FALSE);
	END_IF
END_IF
(* Check timer *)
IF Timer.Q THEN
	TCount:=0;							(* One hour is elapsed *)
	IF TCount<Plant_MaxWaterLoss THEN
		Status_Log:=0;
	END_IF
END_IF
END_FUNCTION_BLOCK
ACTION AddLogData:
Logger.s1:=INSERT('&CTL=',BYTE_TO_STRING(ID),4);
IF ID<10 THEN Logger.s1:=INSERT(Logger.s1,'0',4); END_IF

Logger.s1:=CONCAT(Logger.s1,DWORD_TO_STRING(COUNT));			Logger.s1:=CONCAT(Logger.s1,';');

Logger.s1:=CONCAT(Logger.s1,WORD_TO_STRING(Status_Log));
ADDSTRING(ADR(Logger.TData), ADR(Logger.s1), Logger.TLen);
END_ACTION

(* POU Plant_Objects/obj_MBUS, ST *)
FUNCTION_BLOCK obj_MBUS
(* === M-BUS PROTOCOL INTERFACE ===
   v1.0[16/03/15] - Added interface errors
*)
VAR_INPUT
	(* Settings *)
	ID				: BYTE;
	COM				: BYTE;
	BAUDRATE		: COM_BAUDRATE;
	(* Interface *)
	MBus 			: typMBus;
	MBus_Master 	: FbMBusMaster;
END_VAR
VAR_OUTPUT
	(* Status *)
	Status_Log		: BYTE;
	Status_Vis 		: DWORD;
END_VAR
VAR
	Alarm			: FLT_EVENT;
END_VAR
MBus_Master( bCOMPORT:=COM , enumBAUDRATE:=BAUDRATE , utMBus:=MBus );

(* Check status *)
Alarm(IN:=(MBus.bCOM_ERROR<>0));
IF Alarm.EVH THEN
	LogEv(EL_Alarm,EO_MBUS,ID,1,BYTE_TO_STRING(MBus.bCOM_ERROR));
END_IF
IF Alarm.EVL THEN
	LogEv(EL_Log,EO_MBUS,ID,2,'MBUS_OK');
END_IF

(* Log/visu status *)
   IF Alarm.IN   					THEN Status_Log:=2; Status_Vis:=COLOR_RED;
ELSIF (MBus.bL1_ERROR AND 16#1F)<>0 THEN Status_Log:=1; Status_Vis:=COLOR_YELLOW;
  				 					ELSE Status_Log:=0; Status_Vis:=COLOR_GREEN;
END_IF
END_FUNCTION_BLOCK

(* POU Plant_Objects/obj_MBUS_CTB_SHARKY775, ST *)
FUNCTION_BLOCK obj_MBUS_CTB_SHARKY775
(* === M-BUS CONTABILIZER SHARKY 775 ===
   v1.0[16/03/15] - Error management
*)
VAR_INPUT
	(* Settings *)
	ID				: BYTE;
	ADDRESS			: DWORD;
	Refresh_Period	: TIME:=t#3m;
	(* Controls *)
	Refresh_Auto	: BOOL:=TRUE; (* Enable automatic refresh *)
	Refresh_Now		: BOOL; 	  (* Force an immediate refresh *)
END_VAR
VAR_IN_OUT
	(* Interface *)
	MBUS			: obj_MBUS;
END_VAR
VAR_OUTPUT
	M1				: FbMBus_Heat;
	(* Status *)
	Status_Log		: BYTE;
	Status_Vis 	 	: DWORD;
END_VAR
VAR
	dly 	 	: TON := (PT:=t#5s);
	M1_Start	: BOOL;

	init_st		: BOOL;
	bus_st0		: BYTE;
	dev_st0		: BYTE;

(*	S1			: FbMBusSend;
	S1_Start	: BOOL;*)
(*	C1			: FbUnitConverter; *)

END_VAR
(* Auto refresh timer *)
dly(IN:=NOT (dly.Q OR Refresh_Now OR (NOT Refresh_Auto)));
(* Trigger refresh *)
IF dly.Q OR Refresh_Now THEN
	dly.PT:=Refresh_Period;
	Refresh_Now:=FALSE;
	(* Start reading *)
	M1.dwAdr:= ADDRESS;
	M1.xSND_NKE:=TRUE;
	M1_Start:=TRUE;
END_IF

(* Contabilizer module *)
M1(	utMBus:=MBUS.MBus, xStart:=M1_Start );

(* Extra actions *)
(*C1( utMBus:=MBUS.MBus, xStart:=C1_Start );*)

(* Check status *)
IF NOT init_st OR M1.bError<>bus_st0 OR M1.utMBInfo.bMStatus<>dev_st0 THEN
	init_st:=TRUE;
	bus_st0:=M1.bError; dev_st0:=M1.utMBInfo.bMStatus;
	IF bus_st0<>0 THEN
		LogEv(EL_Alarm,EO_CTB,ID,2,BYTE_TO_STRING(bus_st0));
		Status_Log:=2; Status_Vis:=COLOR_RED;
	ELSE
		IF dev_st0<>0 THEN
			Status_Log:=2; Status_Vis:=COLOR_RED;
			CASE dev_st0 OF
				16#08: LogEv(EL_Alarm,EO_CTB,ID,10,'C-1');
				16#04: LogEv(EL_Alarm,EO_CTB,ID,10,'E-8');
				16#28: LogEv(EL_Alarm,EO_CTB,ID,10,'E-4');
				16#50: LogEv(EL_Alarm,EO_CTB,ID,10,'E-1');
				16#70: LogEv(EL_Alarm,EO_CTB,ID,10,'E-7');
				16#84: LogEv(EL_Alarm,EO_CTB,ID,10,'E-9');
				16#B0: LogEv(EL_Wrn  ,EO_CTB,ID,10,'E-3');
				16#D0: LogEv(EL_Wrn  ,EO_CTB,ID,10,'E-6');
				16#F0: LogEv(EL_Alarm,EO_CTB,ID,10,'Leak');
				16#10: LogEv(EL_Wrn  ,EO_CTB,ID,10,'E-5'); Status_Log:=1; Status_Vis:=COLOR_YELLOW;
			ELSE
				LogEv(EL_Alarm,EO_CTB,ID,10,BYTE_TO_STRING(dev_st0));
			END_CASE
		ELSE
			Status_Log:=0; Status_Vis:=16#20F020;
			LogEv(EL_Log,EO_CTB,ID,1,'');
		END_IF
	END_IF
END_IF
END_FUNCTION_BLOCK
ACTION AddLogData:
Logger.s1:=INSERT('&CTB=',BYTE_TO_STRING(ID),4);
IF ID<10 THEN Logger.s1:=INSERT(Logger.s1,'0',4); END_IF

Logger.s1:=CONCAT(Logger.s1,M1.utFTemp.Value);		Logger.s1:=CONCAT(Logger.s1,';');
Logger.s1:=CONCAT(Logger.s1,M1.utRTemp.Value);		Logger.s1:=CONCAT(Logger.s1,';');
Logger.s1:=CONCAT(Logger.s1,M1.utFlow.Value);		Logger.s1:=CONCAT(Logger.s1,';');
Logger.s1:=CONCAT(Logger.s1,M1.utPower.Value);		Logger.s1:=CONCAT(Logger.s1,';');
Logger.s1:=CONCAT(Logger.s1,M1.utEnergy.Value);		Logger.s1:=CONCAT(Logger.s1,';');

Logger.s1:=CONCAT(Logger.s1,BYTE_TO_STRING(Status_Log));
ADDSTRING(ADR(Logger.TData), ADR(Logger.s1), Logger.TLen);
END_ACTION

(* POU Plant_Objects/obj_MODBUS, ST *)
FUNCTION_BLOCK obj_MODBUS
(* === MODBUS PROTOCOL INTERFACE ===
   v1.1[19/06/15] - Added new VARS allocation and searching
*)
VAR CONSTANT
	VARS_Max	: BYTE := 32;
END_VAR
VAR_INPUT
	(* Settings *)
	ID			: BYTE;
	COM			: BYTE;
	BAUDRATE	: COM_BAUDRATE;
	RS485		: BOOL := FALSE;

	(* Interface *)
	MB_MASTER	: MODBUS_EXTENDED_MASTER;
	MB_Start	: BOOL;
	MB_Query	: typModbusExtendedQuery;
	MB_Resp		: typModbusResponse;
	MB_Lock		: BOOL;

	(* Variables management *)
	VARS_En		: BOOL;
	VARS		: ARRAY [0..VARS_Max] OF typ_MODBUS_VAR;
	VARS_Check	: BOOL;
	VARS_Alarm	: BOOL;

	(* Variables allocation *)
	VAR_Pointer : POINTER TO ARRAY[0..99] OF WORD;
	VAR_Cfg		: POINTER TO typ_MODBUS_VAR;
END_VAR
VAR_OUTPUT
	(* Status *)
	Status_Log	: BYTE;
	Status_Vis	: DWORD;
END_VAR
VAR
	sta         : BYTE :=0;
	i			: BYTE;
	j			: BYTE;
	Alarm		: FLT_EVENT;
	
	VarTmr		: TON := (PT:=T#1s);
	VarSta		: BYTE; (* Status *)
	VarCnt		: BYTE; (* Scan counter *)
	VarRetry	: BYTE;
	VarAlarm	: BYTE; (* Last variable with errors *)
END_VAR
MB_MASTER(ENABLE:=TRUE,	ASCII_Mode:=FALSE, bCOM_PORT:=COM, cbCOM_BAUDRATE:=BAUDRATE, cpCOM_PARITY:=PARITY_NO,
		csCOM_STOPBITS:=STOPBITS_1,	cbsCOM_BYTESIZE:=BS_8, cfCOM_FLOW_CONTROL:=SEL(RS485,NO_FLOW_CONTROL,HALFDUPLEX),
		tTIME_OUT:=t#500ms,	StartFunction:=MB_Start, ExtQuery:=MB_Query, Response:=MB_Resp);

(* Process variable management *)
IF VARS_En THEN VARS_Process(); END_IF

(* Check status *)
Alarm(IN:=(MB_MASTER.bInterfaceError<>0));
IF Alarm.EVH THEN
	LogEv(SEL(MB_MASTER.bInterfaceError<>3,EL_Wrn,EL_Alarm),EO_MODBUS,ID,1,BYTE_TO_STRING(MB_MASTER.bInterfaceError));
END_IF
IF Alarm.EVL THEN								(* Trigger a fall edge: MODBUS back working *)
	LogEv(EL_Log,EO_MODBUS,ID,2,'MODBUS_OK');
END_IF

(* Log/visu status *)
   IF Alarm.IN   THEN Status_Log:=2; Status_Vis:=COLOR_RED;
ELSIF Vars_Alarm THEN Status_Log:=1; Status_Vis:=COLOR_YELLOW;
  				 ELSE Status_Log:=0; Status_Vis:=COLOR_GREEN;
END_IF
END_FUNCTION_BLOCK
ACTION VAR_Search:
(* Search VAR with specific pointer if not found return first free VAR
	[Last VAR is not active... used as safe area...] 
*)
j:=VARS_Max;
FOR i := 0 TO VARS_Max-1 DO
	IF VARS[i].Variable=0 AND j>i THEN j:=i; END_IF
	IF VARS[i].Variable=VAR_Pointer THEN
		VAR_Cfg:=ADR(VARS[i]);
		RETURN;
	END_IF
END_FOR
VAR_Cfg:=ADR(VARS[j]);
END_ACTION
ACTION VARS_Process:
(* Update var timers *)
VarTmr(IN:=(NOT VarTmr.Q));
IF VarTmr.Q THEN
	FOR i := 0 TO VARS_Max DO
		IF VARS[i].Refresh_Cnt>0 THEN VARS[i].Refresh_Cnt:=VARS[i].Refresh_Cnt-1; END_IF
	END_FOR
	VARS_Check:=TRUE;
END_IF


(* Process status *)
CASE VarSta OF
	0: (* === Init *)
		VarCnt:=0;
		VarSta:=1;

	1: (* === Wait check signal *)
		IF VARS_Check THEN				(* Decremented "Refresh_Cnt" *)
			VARS_Check:=FALSE;
			VarCnt:=0;
			VarSta:=2;
		END_IF

	2: (* === Check loop *)
		IF NOT (MB_Lock OR MB_Start) THEN
			WHILE VarCnt<=(VARS_Max-1) AND VarSta=2 DO
				(* Check only active vars *)
				IF VARS[VarCnt].Variable<>0 THEN			(* "Variable" is a pointer to word, so if 0 no address *)
					(* Check var auto-refresh on timer checks *)
					IF VARS[VarCnt].Refresh_Time>0 AND VARS[VarCnt].Refresh_Cnt=0 THEN
						VARS[VarCnt].Refresh_Cnt:=VARS[VarCnt].Refresh_Time;
						VarSta:=3;
					END_IF
					(* Check refresh for change or request *)
					CASE VARS[VarCnt].FunCode OF
						5,6,15,16: (* Write functions *)
							IF VARS[VarCnt].Variable_Size=1 THEN
								IF VARS[VarCnt].Variable^<>VARS[VarCnt].Variable_Mirror THEN
									VARS[VarCnt].Variable_Mirror:=VARS[VarCnt].Variable^;
									VarSta:=3;
								END_IF
							ELSE
								IF VARS[VarCnt].Variable_Mirror<>0 THEN
									VARS[VarCnt].Variable_Mirror:=0;
									VarSta:=3;
								END_IF
							END_IF
						1,2,3,4: (* Read functions *)
							IF VARS[VarCnt].Variable_Mirror<>0 THEN
								VARS[VarCnt].Variable_Mirror:=0;
								VarSta:=3;
							END_IF
					END_CASE
				END_IF
				(* Process query *)
				IF VarSta=3 THEN
					MB_Lock:=TRUE;
					MB_Query.SlaveAddress:=VARS[VarCnt].SlaveAddress;
					MB_Query.FunctionCode:=VARS[VarCnt].FunCode;
					CASE VARS[VarCnt].FunCode OF
						16#5,16#6,16#F,16#10:
							MB_Query.Read_Quantity:=0;
							MB_Query.Read_StartAddress:=0;
							MB_Query.Write_StartAddress:=VARS[VarCnt].FunAddress;
							MB_Query.Write_Quantity:=VARS[VarCnt].Variable_Size;
							IF VARS[VarCnt].Variable_Size=200 THEN
								COPY_32SWAP16(VARS[VarCnt].Variable, ADR(MB_Query.Write_Data[0]));
							ELSIF VARS[VarCnt].Variable_Size>1 THEN
								MEMCPY(VARS[VarCnt].Variable, ADR(MB_Query.Write_Data[0]), 2*VARS[VarCnt].Variable_Size);
							ELSE
								MB_Query.Write_Data[0]:=VARS[VarCnt].Variable^;
							END_IF
						16#1,16#2,16#3,16#4:
							MB_Query.Read_StartAddress:=VARS[VarCnt].FunAddress;
							IF VARS[VarCnt].Variable_Size=200 THEN MB_Query.Read_Quantity:=2; ELSE
							  MB_Query.Read_Quantity:=VARS[VarCnt].Variable_Size;
							END_IF
							MB_Query.Write_StartAddress:=0;
							MB_Query.Write_Quantity:=0;
					END_CASE
					VarRetry:=0;
					MB_Start:=TRUE;
				ELSE
					VarCnt:=VarCnt+1;
				END_IF
			END_WHILE
			(* Check loop completed -> no actions *)
			IF VarSta=2 THEN VarSta:=1; END_IF
		END_IF

	3: (* === Wait & process MB response *)
		IF NOT MB_Start THEN
			IF MB_MASTER.MB_Error=0 THEN
				CASE VARS[VarCnt].FunCode OF
					1,2,3,4:
						IF VARS[VarCnt].Variable_Size=200 THEN
							COPY_32SWAP16(ADR(MB_Resp.Data), VARS[VarCnt].Variable);
						ELSIF VARS[VarCnt].Variable_Size>1 THEN
							MEMCPY(ADR(MB_Resp.Data), VARS[VarCnt].Variable, 2*VARS[VarCnt].Variable_Size);
						ELSE
							VARS[VarCnt].Variable^:=MB_Resp.Data[0];
						END_IF
				END_CASE
				MB_Lock:=FALSE;
				(* Signal error recovery *)
				IF VARS_Alarm=TRUE AND VarCnt=VarAlarm THEN
					LogEv(EL_Wrn,EO_MODBUS,ID,5,'');
					VARS_Alarm:=FALSE;
				END_IF
				(* Next var *)
				VarCnt:=VarCnt+1;
				VarSta:=2;
			ELSE
				IF VarRetry<3 THEN
					VarRetry:=VarRetry+1;
					MB_Start:=TRUE;
				ELSE
					MB_Lock:=FALSE;
					(* Signal error *)
					IF VARS_Alarm=FALSE THEN
						LogEv(EL_Wrn,EO_MODBUS,ID,3,INT_TO_STRING(MB_MASTER.MB_Error));
						VARS_Alarm:=TRUE;
						VarAlarm:=VarCnt-1;
					END_IF
					(* Next var *)
					VarCnt:=VarCnt+1;
					VarSta:=2;
				END_IF
			END_IF
		END_IF

ELSE
	VarSta:=0;
END_CASE
END_ACTION

(* POU Plant_Objects/obj_MODBUS_CIR, ST *)
FUNCTION_BLOCK obj_MODBUS_CIR
VAR CONSTANT
	WAIT_STATE		:	BYTE := 0;
	PUMP_STATUS		:	BYTE := 1;
	PUMP_DATA		:	BYTE := 2;
	PUMP_ALARMS		:	BYTE := 3;
	PUMP_END_READ	:	BYTE := 4;
	CIR_ON_OFF		:	BYTE := 90;
	CIR_ON_OFF_CHECK:	BYTE := 91;
	CIR_END_WRITE	:	BYTE := 92;
	ERROR_STATE		:	BYTE := 100;
END_VAR
VAR_INPUT
	ID		:	BYTE;
	Address :	BYTE;		(* Pump address *)

	(* Physical inputs *)
	CIR_RUN_REQ		: BOOL; (* External run request (no heat or cold requested) *)
	CIR_STOP_REQ	: BOOL; (* External stop request (has priority over RUN signals!) *)

	Pump_AL			: BOOL; (* Alarm input signal *)
	Pump_AUTO		: BOOL;	(* Automatic/Manual input *)

	(* Controls *)
	OnOff		: 	BOOL;
	InitOK		:	BOOL;

	(* Timings *)
	OnDelay		:	TIME;
	OffDelay	:	TIME;

	(* Modbus *)
	Refresh_Now	:	BOOL;	(* Start immediately modbus state machine *)
	retryErrMax	:	BYTE := 2;

	(* Riferimento Velocità da remoto arriva dall'esterno e mi otimizza la portata sulla mandata acqua principale *)

	VelocitaRichiesta:INT;


END_VAR
VAR_IN_OUT
	ModBus		:	obj_MODBUS;
END_VAR
VAR_OUTPUT
	Ctrl_Run	:	BOOL;		(* Logical status of the device: 0: Not running (switched off), 1: running *)
	Run			:	BOOL;		(* Real status *)

	Status_Log	:	WORD;
	Status_Vis	:	DWORD;
END_VAR
VAR
	Pump_En		:	WORD;

	(* Filters *)
	fPump_AL	:	FLT_TAP := (INITEV:=FALSE);
	fPump_ST	:	FLT_TAP := (INITEV:=FALSE);
	fPump_En	:	FLT_EVENT;
	fCIR_AUTO	:	FLT_TAP;
	fStatus		:	FLT_EVENT;
	fStatusFault:	BOOL;

	(* Timer manage switch on/off delay *)
	Delay		: 	TONOF;

	(* CIR data structure *)
	DataPump	:	typ_MODBUS_CIR;

	(* Modbus variables *)
	state		:	BYTE;
	retry		:	BYTE;
	retryErr	:	BYTE;
	ReadTmr		:	TON := (PT:=T#5s);
	fModbusAlr	: 	BOOL;

	(* Alarm and Warning counters *)
	AlarmCtr	:	BYTE;
	WarningCtr	:	BYTE;

	(* Filers on alarms and faults *)
	AlarmHw		:	FLT_TAP;(* := (INITEV:=FALSE);*)
	Alarm		:	FLT_EVENT := (INITEV:=FALSE);
	Inverter	:	FLT_EVENT := (INITEV:=FALSE);
	ModbusAlr	:	FLT_EVENT := (INITEV:=FALSE);

	OldAlarm	:	WORD;


	TimeOutModBus: TON;

END_VAR
Init();

(* Check alarm and warning for both pumps *)
CheckFault();

PumpManager();

(* State machine to read pump parameters *)
Stm();

IF AlarmCtr>0 THEN
	Status_Log := 2;
	Status_Vis := COLOR_RED;
ELSIF WarningCtr>0 OR fPump_ST.OUT THEN
	Status_Log := 1;
	Status_Vis := COLOR_YELLOW;
ELSE
	Status_Log := 0;
	Status_Vis := COLOR_GREEN;
END_IF
END_FUNCTION_BLOCK
ACTION AddLogData:
Logger.s1:=INSERT('&CIRM=',BYTE_TO_STRING(ID),5);
IF ID<10 THEN Logger.s1:=INSERT(Logger.s1,'0',5); END_IF

(* NB If value equals 0x7FFF (32767) this means that it is not available -->> Change it to 0 *)
Logger.s1:=CONCAT(Logger.s1,WORD_TO_STRING(DataPump.PumpStatus));											Logger.s1:=CONCAT(Logger.s1,';');
Logger.s1:=CONCAT(Logger.s1,INT_TO_STRING(SEL(DataPump.PumpBoardTemp=16#7FFF,DataPump.PumpBoardTemp,0)));	Logger.s1:=CONCAT(Logger.s1,';');
Logger.s1:=CONCAT(Logger.s1,WORD_TO_STRING(SEL(DataPump.PumpVoltage=16#7FFF,DataPump.PumpVoltage,0)));		Logger.s1:=CONCAT(Logger.s1,';');
Logger.s1:=CONCAT(Logger.s1,WORD_TO_STRING(SEL(DataPump.PumpCurrent=16#7FFF,DataPump.PumpCurrent,0)));		Logger.s1:=CONCAT(Logger.s1,';');
Logger.s1:=CONCAT(Logger.s1,WORD_TO_STRING(SEL(DataPump.PumpPower=16#7FFF,DataPump.PumpPower,0)));			Logger.s1:=CONCAT(Logger.s1,';');
Logger.s1:=CONCAT(Logger.s1,WORD_TO_STRING(SEL(DataPump.PumpRPM=16#7FFF,DataPump.PumpRPM,0)));				Logger.s1:=CONCAT(Logger.s1,';');
Logger.s1:=CONCAT(Logger.s1,WORD_TO_STRING(SEL(DataPump.PumpHead=16#7FFF,DataPump.PumpHead,0)));				Logger.s1:=CONCAT(Logger.s1,';');
Logger.s1:=CONCAT(Logger.s1,WORD_TO_STRING(SEL(DataPump.PumpFlow=16#7FFF,DataPump.PumpFlow,0)));				Logger.s1:=CONCAT(Logger.s1,';');
Logger.s1:=CONCAT(Logger.s1,WORD_TO_STRING(SEL(DataPump.PumpLiqTemp=16#7FFF,DataPump.PumpLiqTemp,0)));		Logger.s1:=CONCAT(Logger.s1,';');
Logger.s1:=CONCAT(Logger.s1,DWORD_TO_STRING(SEL(DataPump.PumpOpTime=16#7FFF,DataPump.PumpOpTime,0)));		Logger.s1:=CONCAT(Logger.s1,';');

Logger.s1:=CONCAT(Logger.s1,WORD_TO_STRING(Status_Log));
Logger.s1:=CONCAT(Logger.s1,';');

Logger.s1:=CONCAT(Logger.s1,SEL(DataPump.PumpFault,'0','100'));
Logger.s1:=CONCAT(Logger.s1,';');
Logger.s1:=CONCAT(Logger.s1,SEL(CIR_RUN_REQ,'0','100'));
Logger.s1:=CONCAT(Logger.s1,';');
Logger.s1:=CONCAT(Logger.s1,SEL(CIR_STOP_REQ,'0','100'));


ADDSTRING(ADR(Logger.TData), ADR(Logger.s1), Logger.TLen);
END_ACTION
ACTION CheckFault:
(*** WARNINGS ***)

(* Verify ModBus error	*)
ModbusAlr(IN:=fModbusAlr);

IF ModbusAlr.EVH THEN
	LogEv(EL_Wrn,EO_CIRM,ID,13,SEL(ModBus.MB_MASTER.MB_Error<>0,'0','1'));
	WarningCtr := WarningCtr + 1;
END_IF

IF ModbusAlr.EVL THEN WarningCtr := SEL(WarningCtr=0, WarningCtr-1, 0); END_IF


(*** ALARMS ***)

(* Hardware alarm (physical input *)
AlarmHw(IN:=Pump_AL);

IF AlarmHw.EVH THEN
	LogEv(EL_Alarm,EO_CIRM,ID,3,'CIR_Alarm');
	AlarmCtr := AlarmCtr + 1;
END_IF

IF AlarmHw.EVL THEN
	LogEv(EL_Log,EO_CIRM,ID,4,'CIR_Alarm_Recovered');
	AlarmCtr := SEL(AlarmCtr=0, AlarmCtr-1, 0);
END_IF

(*
(* General alarm (read by Modbus) *)
Alarm(IN:=(DataPump.PumpAlarm[0] <> OldAlarm));

IF Alarm.EVH THEN
	IF DataPump.PumpAlarm[0] = 0 THEN
		LogEv(EL_Log,EO_CIRM,ID,12,'Alarm_Recovered');
		AlarmCtr := SEL(AlarmCtr=0, AlarmCtr-1, 0);
	ELSE
		LogEv(EL_Alarm,EO_CIRM,ID,11,WORD_TO_STRING(DataPump.PumpAlarm[0]));
		AlarmCtr := AlarmCtr + 1;
	END_IF

	OldAlarm := DataPump.PumpAlarm[0];
END_IF


(* Inverter pump error *)
Inverter(IN:=DataPump.PumpFault);

IF Inverter.EVH THEN
	LogEv(EL_Alarm,EO_CIRM,ID,9,'Inverter_Fault');
	AlarmCtr := AlarmCtr + 1;
END_IF

IF Inverter.EVL THEN
	LogEv(EL_Alarm,EO_CIRM,ID,10,'Inverter_Fault_Recovered');
		AlarmCtr := SEL(AlarmCtr=0, AlarmCtr-1, 0);
END_IF

*)
END_ACTION
ACTION Init:
IF NOT InitOK THEN

	Delay.PT_OF := SEL(OffDelay=T#0ms, OffDelay, Plant_CirOffDelay);
	Delay.PT_ON := SEL(OnDelay=T#0ms, OnDelay, Plant_CirOnDelay) + WORD_TO_TIME(1000*ID);

	ReadTmr.PT := WORD_TO_TIME(1000*ID);	(* 1s delay between reads of 2 different double CIRs *)

	Pump_En := 1;
	Refresh_Now := TRUE;

	InitOK := TRUE;

END_IF
END_ACTION
ACTION PumpManager:
(*** Verify Status ***)
IF Pump_AUTO THEN
	IF (Pump_En=1 AND DataPump.PumpStatus=2) OR (Pump_En=0 AND DataPump.PumpStatus=0) THEN fStatusFault := TRUE;
	ELSE fStatusFault := FALSE;
	END_IF
END_IF

fPump_ST(IN:=fStatusFault);

IF fPump_ST.EVH THEN
	LogEv(SEL(Pump_En=1,EL_Alarm,EL_Wrn),EO_CIRM,ID,SEL(Pump_En=1,5,6),'');
	WarningCtr := WarningCtr + 1;
END_IF

IF fPump_ST.EVL THEN WarningCtr := SEL(WarningCtr=0, WarningCtr-1, 0); END_IF

(* Verify if in Auto or Manual mode *)
fCIR_AUTO(IN:=Pump_AUTO);

(* Automatic *)
IF fCIR_AUTO.EVH THEN
	LogEv(EL_Log,EO_CIRM,ID,8,'CIR_Auto');
	WarningCtr := SEL(WarningCtr=0, WarningCtr-1, 0);

	Refresh_Now := TRUE;
END_IF

(* Manual -> Keep switched on *)
IF fCIR_AUTO.EVL THEN
	LogEv(EL_Wrn,EO_CIRM,ID,7,'CIR_Manual');
	WarningCtr := WarningCtr + 1;

	Pump_En := 0;
	Refresh_Now := TRUE;
END_IF

(* Verify if OnOff is changed *)
Ctrl_Run := OnOff;

(* Check switch on or switch off delay *)
Delay(IN:=Ctrl_Run);

IF Pump_AUTO THEN
	(* If priority request *)
	IF CIR_STOP_REQ THEN Pump_En := 1;
	ELSIF CIR_RUN_REQ THEN Pump_En := 0;
	ELSE Pump_En := BOOL_TO_WORD(NOT Delay.OUT);
	END_IF

	(* Set RUN signal (for external objects) *)
	IF AlarmHw.OUT THEN
		Run:=FALSE;
	ELSE
		Run:=SEL(Pump_En=1,TRUE,FALSE);
	END_IF
END_IF

(* Check if a pump enable update (modbus write) is requested *)
fPump_En(IN:=(Pump_En=1));

IF fPump_En.EVH OR fPump_En.EVL THEN
	Refresh_Now := TRUE;
END_IF
END_ACTION
ACTION Stm:
CASE state OF
	WAIT_STATE:	(* Refresh time manager *)
		ReadTmr(IN:=NOT ReadTmr.Q);
		TimeOutModBus(In:=state<>0,PT:=t#5s);
		IF ReadTmr.Q OR Refresh_Now AND NOT MODBUS.MB_Lock THEN
			state := PUMP_STATUS;
			ReadTmr.PT := T#1m0s;  (* moreno *)
			Refresh_Now := FALSE;
			Modbus.MB_Lock := TRUE;
		END_IF

	(**** READ CIR PARAMETERS ****)

	PUMP_STATUS:	(* Status and Fault *)
		Modbus.MB_Lock := TRUE;
		Modbus.MB_Query.SlaveAddress := Address;
		Modbus.MB_Query.FunctionCode := 4;
		ModBus.MB_Query.Read_StartAddress := 201;
		ModBus.MB_Query.Read_Quantity := 2;
		ModBus.MB_Start := TRUE;

		state := PUMP_DATA;


	PUMP_DATA:	(* Pump data *)
		IF NOT ModBus.MB_Start  AND ModBus.MB_Resp.SlaveAddress=Address  THEN
			IF ModBus.MB_MASTER.MB_Error<>0 THEN (*OR ModBus.MB_MASTER.MB_Error<>0 THEN*)
				state := ERROR_STATE;
			ELSE
				DataPump.PumpStatus := ModBus.MB_Resp.Data[0];
				DataPump.PumpFault	:= WORD_TO_BOOL(ModBus.MB_Resp.Data[1]);

				ModBus.MB_Query.Read_StartAddress := 210;
				ModBus.MB_Query.Read_Quantity := 12;
				ModBus.MB_Start := TRUE;

				state := PUMP_ALARMS;
			END_IF
		END_IF

	PUMP_ALARMS: (* Historical alarms *)
		IF NOT ModBus.MB_Start  AND ModBus.MB_Resp.SlaveAddress=Address  THEN

			IF ModBus.MB_MASTER.MB_Error<>0 THEN (*OR ModBus.MB_MASTER.MB_Error<>0 THEN*)
				state := ERROR_STATE;
			ELSE
				DataPump.PumpBoardTemp 	:= WORD_TO_INT(ModBus.MB_Resp.Data[0]);
				DataPump.PumpVoltage	:= ModBus.MB_Resp.Data[2];
				DataPump.PumpCurrent	:= ModBus.MB_Resp.Data[3];
				DataPump.PumpRPM		:= ModBus.MB_Resp.Data[5];
				DataPump.PumpPower		:= ModBus.MB_Resp.Data[6];
				DataPump.PumpOpTime		:= BUILD_16TO32(ADR(ModBus.MB_Resp.Data[7]));
				DataPump.PumpHead		:= ModBus.MB_Resp.Data[9];
				DataPump.PumpFlow		:= ModBus.MB_Resp.Data[10];
				DataPump.PumpLiqTemp	:= WORD_TO_INT(ModBus.MB_Resp.Data[11]);


				ModBus.MB_Query.Read_StartAddress := 230;
				ModBus.MB_Query.Read_Quantity := 1;(*15;*)
				ModBus.MB_Start := TRUE;

				state := PUMP_END_READ;
			END_IF
		END_IF

	PUMP_END_READ:	(* Read alarms *)
		IF NOT ModBus.MB_Start  AND ModBus.MB_Resp.SlaveAddress=Address  THEN
			IF ModBus.MB_MASTER.MB_Error<>0 THEN (*OR ModBus.MB_MASTER.MB_Error<>0 THEN*)
				state := ERROR_STATE;
			ELSE
				DataPump.PumpAlarm[0] := ModBus.MB_Resp.Data[0];	(* Read just last (most recent) alarm *)
				(*DataPump.PumpAlarm[1] := ModBus.MB_Resp.Data[1];
				DataPump.PumpAlarm[2] := ModBus.MB_Resp.Data[2];
				DataPump.PumpAlarm[3] := ModBus.MB_Resp.Data[3];
				DataPump.PumpAlarm[4] := ModBus.MB_Resp.Data[4];
				DataPump.PumpAlarm[5] := ModBus.MB_Resp.Data[5];
				DataPump.PumpAlarm[6] := ModBus.MB_Resp.Data[6];
				DataPump.PumpAlarm[7] := ModBus.MB_Resp.Data[7];
				DataPump.PumpAlarm[8] := ModBus.MB_Resp.Data[8];
				DataPump.PumpAlarm[9] := ModBus.MB_Resp.Data[9];
				DataPump.PumpAlarm[10] := ModBus.MB_Resp.Data[10];
				DataPump.PumpAlarm[11] := ModBus.MB_Resp.Data[11];
				DataPump.PumpAlarm[12] := ModBus.MB_Resp.Data[12];
				DataPump.PumpAlarm[13] := ModBus.MB_Resp.Data[13];
				DataPump.PumpAlarm[14] := ModBus.MB_Resp.Data[14];*)

				state := CIR_ON_OFF;

			END_IF
		END_IF

	(**** WRITE ON/OFF REGISTER AND VERIFY RIGHT SETTING ****)
	CIR_ON_OFF:	(* Pump On/off *)

		Modbus.MB_Query.SlaveAddress := Address;
		Modbus.MB_Query.FunctionCode := 6;
		ModBus.MB_Query.Write_StartAddress := 109;
		ModBus.MB_Query.Write_Quantity := 2;
		ModBus.MB_Query.Write_Data[0] := VelocitaRichiesta;
		ModBus.MB_Query.Write_Data[1] := Pump_En;
		ModBus.MB_Start := TRUE;

	state := CIR_END_WRITE;

	CIR_END_WRITE:
		IF NOT ModBus.MB_Start THEN
			IF ModBus.MB_MASTER.bInterfaceError<>0 THEN (*OR ModBus.MB_MASTER.MB_Error<>0 THEN*)
				state := ERROR_STATE;
			ELSE
				IF fModbusAlr THEN fModbusAlr := FALSE; END_IF

				ModBus.MB_Lock := FALSE;
				retryErr := 0;
				retry := 0;
				state := WAIT_STATE;
			END_IF
		END_IF


	(**** CHECK MODBUS ERROR ****)
	ERROR_STATE: 	(* Release MODBUS *)
			MODBUS.MB_Lock:=FALSE;

			(* Retries *)
			retry:=retry+1;
			IF retry>3 THEN
				retry:=0;

				(* Verify if slave is dead *)
				IF retryErr < retryErrMaX THEN
					retryErr := retryErr + 1;
				ELSE
					fModbusAlr := TRUE;
				END_IF

				Refresh_Now := FALSE;
			END_IF

			state:=WAIT_STATE;
END_CASE





(* Controllo Time Out Ciclo ModBus *)

TimeOutModBus(In:=state<>0,PT:=t#5s);
IF TimeOutModBus.Q THEN
	State:=0;
	Refresh_Now:=TRUE;  (* Rilancio la lettura del nodo *)
	IF MODBUS.MB_Lock=TRUE THEN MODBUS.MB_Lock:=FALSE;END_IF
END_IF
END_ACTION

(* POU Plant_Objects/obj_MODBUS_CIR_DAB, ST *)
FUNCTION_BLOCK obj_MODBUS_CIR_DAB
VAR CONSTANT
	WAIT_STATE		:	BYTE := 0;
	PUMP_STATUS		:	BYTE := 1;
	PUMP_DATA		:	BYTE := 2;
	PUMP_ALARMS		:	BYTE := 3;
	PUMP_END_READ	:	BYTE := 4;
	CIR_ON_OFF		:	BYTE := 90;
	CIR_ON_OFF_CHECK:	BYTE := 91;
	CIR_END_WRITE	:	BYTE := 92;
	ERROR_STATE		:	BYTE := 100;
END_VAR
VAR_INPUT
	ID		:	BYTE;
	Address :	BYTE;		(* Pump address *)

	(* Physical inputs *)
	CIR_RUN_REQ		: BOOL; (* External run request (no heat or cold requested) *)
	CIR_STOP_REQ	: BOOL; (* External stop request (has priority over RUN signals!) *)

	Pump_AL			: BOOL; (* Alarm input signal *)
	Pump_AUTO		: BOOL;	(* Automatic/Manual input *)

	(* Controls *)
	OnOff		: 	BOOL;
	InitOK		:	BOOL;

	(* Timings *)
	OnDelay		:	TIME;
	OffDelay	:	TIME;

	(* Modbus *)
	Refresh_Now	:	BOOL;	(* Start immediately modbus state machine *)
	retryErrMax	:	BYTE := 2;

	(* Riferimento Velocità da remoto arriva dall'esterno e mi otimizza la portata sulla mandata acqua principale *)

	VelocitaRichiesta:INT:=100;

END_VAR
VAR_IN_OUT
	ModBus		:	obj_MODBUS;
END_VAR
VAR_OUTPUT
	Ctrl_Run	:	BOOL;		(* Logical status of the device: 0: Not running (switched off), 1: running *)
	Run			:	BOOL;		(* Real status *)

	Status_Log	:	WORD;
	Status_Vis	:	DWORD;
END_VAR
VAR
	Pump_En		:	WORD;

	(* Filters *)
	fPump_AL	:	FLT_TAP := (INITEV:=FALSE);
	fPump_ST	:	FLT_TAP := (INITEV:=FALSE);
	fPump_En	:	FLT_EVENT;
	fCIR_AUTO	:	FLT_TAP;
	fStatus		:	FLT_EVENT;
	fStatusFault:	BOOL;

	(* Timer manage switch on/off delay *)
	Delay		: 	TONOF;

	(* CIR data structure *)
	DataPump	:	typ_MODBUS_CIR;

	(* Modbus variables *)
	state		:	INT;
	retry		:	BYTE;
	retryErr	:	BYTE;
	ReadTmr		:	TON := (PT:=T#5s);
	fModbusAlr	: 	BOOL;

	(* Alarm and Warning counters *)
	AlarmCtr	:	BYTE;
	WarningCtr	:	BYTE;

	(* Filers on alarms and faults *)
	AlarmHw		:	FLT_TAP;(* := (INITEV:=FALSE);*)
	Alarm		:	FLT_EVENT := (INITEV:=FALSE);
	Inverter	:	FLT_EVENT := (INITEV:=FALSE);
	ModbusAlr	:	FLT_EVENT := (INITEV:=FALSE);

	OldAlarm	:	WORD;


	TimeOutModBus: TON;
	ErroreComuModBus: BOOL;

	VerificaFuctionCode: INT;
	VerificaNodoLetto: INT;

	TempoTest:TON;

END_VAR
Init();

(* Check alarm and warning for both pumps *)
CheckFault();

PumpManager();

(* State machine to read pump parameters *)
Stm();

IF AlarmCtr>0 THEN
	Status_Log := 2;
	Status_Vis := COLOR_RED;
ELSIF WarningCtr>0 OR fPump_ST.OUT THEN
	Status_Log := 1;
	Status_Vis := COLOR_YELLOW;
ELSE
	Status_Log := 0;
	Status_Vis := COLOR_GREEN;
END_IF
END_FUNCTION_BLOCK
ACTION AddLogData:
Logger.s1:=INSERT('&CIRM=',BYTE_TO_STRING(ID),5);
IF ID<10 THEN Logger.s1:=INSERT(Logger.s1,'0',5); END_IF

(* NB If value equals 0x7FFF (32767) this means that it is not available -->> Change it to 0 *)
Logger.s1:=CONCAT(Logger.s1,WORD_TO_STRING(DataPump.PumpStatus));											Logger.s1:=CONCAT(Logger.s1,';');
Logger.s1:=CONCAT(Logger.s1,INT_TO_STRING(SEL(DataPump.PumpBoardTemp=16#7FFF,DataPump.PumpBoardTemp,0)));	Logger.s1:=CONCAT(Logger.s1,';');
Logger.s1:=CONCAT(Logger.s1,WORD_TO_STRING(SEL(DataPump.PumpVoltage=16#7FFF,DataPump.PumpVoltage,0)));		Logger.s1:=CONCAT(Logger.s1,';');
Logger.s1:=CONCAT(Logger.s1,WORD_TO_STRING(SEL(DataPump.PumpCurrent=16#7FFF,DataPump.PumpCurrent,0)));		Logger.s1:=CONCAT(Logger.s1,';');
Logger.s1:=CONCAT(Logger.s1,WORD_TO_STRING(SEL(DataPump.PumpPower=16#7FFF,DataPump.PumpPower,0)));			Logger.s1:=CONCAT(Logger.s1,';');
Logger.s1:=CONCAT(Logger.s1,WORD_TO_STRING(SEL(DataPump.PumpRPM=16#7FFF,DataPump.PumpRPM,0)));				Logger.s1:=CONCAT(Logger.s1,';');
Logger.s1:=CONCAT(Logger.s1,WORD_TO_STRING(SEL(DataPump.PumpHead=16#7FFF,DataPump.PumpHead,0)));				Logger.s1:=CONCAT(Logger.s1,';');
Logger.s1:=CONCAT(Logger.s1,WORD_TO_STRING(SEL(DataPump.PumpFlow=16#7FFF,DataPump.PumpFlow,0)));				Logger.s1:=CONCAT(Logger.s1,';');
Logger.s1:=CONCAT(Logger.s1,WORD_TO_STRING(SEL(DataPump.PumpLiqTemp=16#7FFF,DataPump.PumpLiqTemp,0)));		Logger.s1:=CONCAT(Logger.s1,';');
Logger.s1:=CONCAT(Logger.s1,DWORD_TO_STRING(SEL(DataPump.PumpOpTime=16#7FFF,DataPump.PumpOpTime,0)));		Logger.s1:=CONCAT(Logger.s1,';');

Logger.s1:=CONCAT(Logger.s1,WORD_TO_STRING(Status_Log));
Logger.s1:=CONCAT(Logger.s1,';');

Logger.s1:=CONCAT(Logger.s1,SEL(DataPump.PumpFault,'0','100'));
Logger.s1:=CONCAT(Logger.s1,';');
Logger.s1:=CONCAT(Logger.s1,SEL(CIR_RUN_REQ,'0','100'));
Logger.s1:=CONCAT(Logger.s1,';');
Logger.s1:=CONCAT(Logger.s1,SEL(CIR_STOP_REQ,'0','100'));


ADDSTRING(ADR(Logger.TData), ADR(Logger.s1), Logger.TLen);
END_ACTION
ACTION CheckFault:
(*** WARNINGS ***)

(* Verify ModBus error	*)
ModbusAlr(IN:=fModbusAlr);

IF ModbusAlr.EVH THEN
	LogEv(EL_Wrn,EO_CIRM,ID,13,SEL(ModBus.MB_MASTER.MB_Error<>0,'0','1'));
	WarningCtr := WarningCtr + 1;
END_IF

IF ModbusAlr.EVL THEN WarningCtr := SEL(WarningCtr=0, WarningCtr-1, 0); END_IF


(*** ALARMS ***)

(* Hardware alarm (physical input *)
AlarmHw(IN:=Pump_AL);

IF AlarmHw.EVH THEN
	LogEv(EL_Alarm,EO_CIRM,ID,3,'CIR_Alarm');
	AlarmCtr := AlarmCtr + 1;
END_IF

IF AlarmHw.EVL THEN
	LogEv(EL_Log,EO_CIRM,ID,4,'CIR_Alarm_Recovered');
	AlarmCtr := SEL(AlarmCtr=0, AlarmCtr-1, 0);
END_IF

(*
(* General alarm (read by Modbus) *)
Alarm(IN:=(DataPump.PumpAlarm[0] <> OldAlarm));

IF Alarm.EVH THEN
	IF DataPump.PumpAlarm[0] = 0 THEN
		LogEv(EL_Log,EO_CIRM,ID,12,'Alarm_Recovered');
		AlarmCtr := SEL(AlarmCtr=0, AlarmCtr-1, 0);
	ELSE
		LogEv(EL_Alarm,EO_CIRM,ID,11,WORD_TO_STRING(DataPump.PumpAlarm[0]));
		AlarmCtr := AlarmCtr + 1;
	END_IF

	OldAlarm := DataPump.PumpAlarm[0];
END_IF


(* Inverter pump error *)
Inverter(IN:=DataPump.PumpFault);

IF Inverter.EVH THEN
	LogEv(EL_Alarm,EO_CIRM,ID,9,'Inverter_Fault');
	AlarmCtr := AlarmCtr + 1;
END_IF

IF Inverter.EVL THEN
	LogEv(EL_Alarm,EO_CIRM,ID,10,'Inverter_Fault_Recovered');
		AlarmCtr := SEL(AlarmCtr=0, AlarmCtr-1, 0);
END_IF

*)
END_ACTION
ACTION Init:
IF NOT InitOK THEN

	Delay.PT_OF := SEL(OffDelay=T#0ms, OffDelay, Plant_CirOffDelay);
	Delay.PT_ON := SEL(OnDelay=T#0ms, OnDelay, Plant_CirOnDelay) + WORD_TO_TIME(1000*ID);

	ReadTmr.PT := WORD_TO_TIME(1000*ID);	(* 1s delay between reads of 2 different double CIRs *)

	Pump_En := 1;
	Refresh_Now := TRUE;

	InitOK := TRUE;

END_IF
END_ACTION
ACTION PumpManager:
(*** Verify Status ***)
IF Pump_AUTO THEN
	IF (Pump_En=1 AND DataPump.PumpStatus=2) OR (Pump_En=0 AND DataPump.PumpStatus=0) THEN fStatusFault := TRUE;
	ELSE fStatusFault := FALSE;
	END_IF
END_IF

fPump_ST(IN:=fStatusFault);

IF fPump_ST.EVH THEN
	LogEv(SEL(Pump_En=1,EL_Alarm,EL_Wrn),EO_CIRM,ID,SEL(Pump_En=1,5,6),'');
	WarningCtr := WarningCtr + 1;
END_IF

IF fPump_ST.EVL THEN WarningCtr := SEL(WarningCtr=0, WarningCtr-1, 0); END_IF

(* Verify if in Auto or Manual mode *)
fCIR_AUTO(IN:=Pump_AUTO);

(* Automatic *)
IF fCIR_AUTO.EVH THEN
	LogEv(EL_Log,EO_CIRM,ID,8,'CIR_Auto');
	WarningCtr := SEL(WarningCtr=0, WarningCtr-1, 0);

	Refresh_Now := TRUE;
END_IF

(* Manual -> Keep switched on *)
IF fCIR_AUTO.EVL THEN
	LogEv(EL_Wrn,EO_CIRM,ID,7,'CIR_Manual');
	WarningCtr := WarningCtr + 1;

	Pump_En := 0;
	Refresh_Now := TRUE;
END_IF

(* Verify if OnOff is changed *)
Ctrl_Run := OnOff;

(* Check switch on or switch off delay *)
Delay(IN:=Ctrl_Run);

IF Pump_AUTO THEN
	(* If priority request *)
	IF CIR_STOP_REQ THEN Pump_En := 1;
	ELSIF CIR_RUN_REQ THEN Pump_En := 0;
	ELSE Pump_En := BOOL_TO_WORD(NOT Delay.OUT);
	END_IF

	(* Set RUN signal (for external objects) *)
	IF AlarmHw.OUT THEN
		Run:=FALSE;
	ELSE
		Run:=SEL(Pump_En=1,TRUE,FALSE);
	END_IF
END_IF

(* Check if a pump enable update (modbus write) is requested *)
fPump_En(IN:=(Pump_En=1));

IF fPump_En.EVH OR fPump_En.EVL THEN
	Refresh_Now := TRUE;
END_IF
END_ACTION
ACTION Stm:
CASE state OF
	0:	(* Refresh time manager *)
		ReadTmr(IN:=NOT ReadTmr.Q);
		TimeOutModBus(In:=state<>0,PT:=t#5s);
		(*A tempo interrogo il nodo sempre che non ci sia qualcuno che lo sta interrogando in quel momento *)

		IF (ReadTmr.Q AND NodoDaInterrogare=Address )OR Refresh_Now AND NOT InibiscoModbus THEN
			state := 10;
			ReadTmr.PT := T#10s;  (* moreno *)
			Refresh_Now := FALSE;
			InibiscoModbus := TRUE;
		END_IF

	(**** READ CIR PARAMETERS ****)

	10:	(* richiedo lettura stato Pompa  *)

		Modbus.MB_Query.SlaveAddress := Address;
		Modbus.MB_Query.FunctionCode := 3;
		ModBus.MB_Query.Read_StartAddress := 201;
		ModBus.MB_Query.Read_Quantity := 2;
		ModBus.MB_Start := TRUE;

		state := 20;

	20:	(* Ripsosta *)
		IF NOT ModBus.MB_Start   THEN
			VerificaFuctionCode:=ModBus.MB_Resp.FunctionCode;
			VerificaNodoLetto:=ModBus.MB_Resp.SlaveAddress;

			IF ModBus.MB_MASTER.MB_Error<>0 THEN (*OR ModBus.MB_MASTER.MB_Error<>0 THEN*)
				state := 300;
			ELSE
				DataPump.PumpStatus := ModBus.MB_Resp.Data[0];  				(*0 - Pompa spenta / 1- Stato di carica / 2- Pompa in moto *)	 																	(*0 - Pompa spenta / 1- Stato di carica / 2- Pompa in moto *)
				DataPump.PumpFault	:= WORD_TO_BOOL(ModBus.MB_Resp.Data[1]); 	(* 0- Ok / 1- Fault *)

				ModBus.MB_Query.Read_StartAddress := 210; (* richiedo lettura stato Pompa Altri PAramentri *)
				ModBus.MB_Query.Read_Quantity := 12;
				ModBus.MB_Start := TRUE;

				state := 30;
			END_IF
		END_IF

	30: (* Ripsota Altri paramenti Stato Pompa *)
		IF NOT ModBus.MB_Start  THEN

			IF ModBus.MB_MASTER.MB_Error<>0 THEN (*OR ModBus.MB_MASTER.MB_Error<>0 THEN*)
				state := 300;
			ELSE
				DataPump.PumpBoardTemp 	:= WORD_TO_INT(ModBus.MB_Resp.Data[0]);
				DataPump.PumpVoltage	:= ModBus.MB_Resp.Data[2];
				DataPump.PumpCurrent	:= ModBus.MB_Resp.Data[3];
				DataPump.PumpRPM		:= ModBus.MB_Resp.Data[5];
				DataPump.PumpPower		:= ModBus.MB_Resp.Data[6];
				DataPump.PumpOpTime		:= BUILD_16TO32(ADR(ModBus.MB_Resp.Data[7]));
				DataPump.PumpHead		:= ModBus.MB_Resp.Data[9];
				DataPump.PumpFlow		:= ModBus.MB_Resp.Data[10];
				DataPump.PumpLiqTemp	:= WORD_TO_INT(ModBus.MB_Resp.Data[11]);


				ModBus.MB_Query.Read_StartAddress := 230; (* Lettura Allarmi presenti nella pompa *)
				ModBus.MB_Query.Read_Quantity := 1;(*15;*)
				ModBus.MB_Start := TRUE;

				state := 40;
			END_IF
		END_IF

	40:	(* Read alarms *)
		IF NOT ModBus.MB_Start   THEN
			IF ModBus.MB_MASTER.MB_Error<>0 THEN (*OR ModBus.MB_MASTER.MB_Error<>0 THEN*)
				state := 300;
			ELSE
				DataPump.PumpAlarm[0] := ModBus.MB_Resp.Data[0];	(* Read just last (most recent) alarm *)
				(*DataPump.PumpAlarm[1] := ModBus.MB_Resp.Data[1];
				DataPump.PumpAlarm[2] := ModBus.MB_Resp.Data[2];
				DataPump.PumpAlarm[3] := ModBus.MB_Resp.Data[3];
				DataPump.PumpAlarm[4] := ModBus.MB_Resp.Data[4];
				DataPump.PumpAlarm[5] := ModBus.MB_Resp.Data[5];
				DataPump.PumpAlarm[6] := ModBus.MB_Resp.Data[6];
				DataPump.PumpAlarm[7] := ModBus.MB_Resp.Data[7];
				DataPump.PumpAlarm[8] := ModBus.MB_Resp.Data[8];
				DataPump.PumpAlarm[9] := ModBus.MB_Resp.Data[9];
				DataPump.PumpAlarm[10] := ModBus.MB_Resp.Data[10];
				DataPump.PumpAlarm[11] := ModBus.MB_Resp.Data[11];
				DataPump.PumpAlarm[12] := ModBus.MB_Resp.Data[12];
				DataPump.PumpAlarm[13] := ModBus.MB_Resp.Data[13];
				DataPump.PumpAlarm[14] := ModBus.MB_Resp.Data[14];*)

				state := 100;

			END_IF
		END_IF

	(**** Dopo La Lettura Scrivo i paramentri ON/OFF e la velocità  ****)
	 100:	(* Pump On/off *)

		Modbus.MB_Query.SlaveAddress := Address;
		Modbus.MB_Query.FunctionCode := 16;
		ModBus.MB_Query.Write_StartAddress := 109;
		ModBus.MB_Query.Write_Quantity :=2;
		ModBus.MB_Query.Write_Data[0] := VelocitaRichiesta;
		ModBus.MB_Query.Write_Data[1] := Pump_En;
		ModBus.MB_Start := TRUE;

		state := 110;

		110:
		IF NOT ModBus.MB_Start THEN
			IF ModBus.MB_MASTER.MB_Error<>0 THEN (*OR ModBus.MB_MASTER.MB_Error<>0 THEN*)
				state := 300;
			ELSE
				IF fModbusAlr THEN fModbusAlr := FALSE; END_IF

				NodoDaInterrogare:=Address+1;
				InibiscoModbus:=FALSE;
				retryErr := 0;
				retry := 0;
				state := 0;
			END_IF
		END_IF


	(**** CHECK MODBUS ERROR ****)
	300: 	(* Release MODBUS *)
			InibiscoModbus:=FALSE;
			(* Retries *)
			retry:=retry+1;
			IF retry>3 THEN
				retry:=0;

				(* Verify if slave is dead *)
				IF retryErr < retryErrMaX THEN
					retryErr := retryErr + 1;
				ELSE
					fModbusAlr := TRUE;
					(* Verify ModBus error	*)

					IF fModbusAlr AND ErroreComuModBus=FALSE THEN
						LogEv(EL_Alarm,EO_CIRDM,ID,13,CONCAT('ErroreModbus_',INT_TO_STRING(ModBus.MB_MASTER.MB_Error)));
						ErroreComuModBus := TRUE;
					END_IF
					IF fModbusAlr=FALSE AND retryErr=0 THEN
						LogEv(EL_Log,EO_CIRDM,ID,14,'ComunicazioneModBus_OK');
							ErroreComuModBus := FALSE;
					(*	WarningCtr := SEL(WarningCtr=0, WarningCtr-1, 0); *)
					END_IF
				END_IF

				END_IF
			Refresh_Now := FALSE;
			NodoDaInterrogare:=Address+1;
			state:=0;
END_CASE





(* Controllo Time Out Ciclo ModBus *)

TimeOutModBus(In:=state<>0,PT:=t#5s);
IF TimeOutModBus.Q THEN
	State:=0;
	Refresh_Now:=TRUE;  (* Rilancio la lettura del nodo *)
	IF MODBUS.MB_Lock=TRUE THEN MODBUS.MB_Lock:=FALSE;END_IF
	IF InibiscoModbus=TRUE THEN InibiscoModbus:=FALSE;END_IF
END_IF
END_ACTION

(* POU Plant_Objects/obj_MODBUS_CIR_DOPPIO_DAB, ST *)
FUNCTION_BLOCK obj_MODBUS_CIR_DOPPIO_DAB
VAR CONSTANT
	WAIT_STATE		:	BYTE := 0;
	PUMP1_STATUS	:	BYTE := 1;
	PUMP1_DATA		:	BYTE := 2;
	PUMP1_ALARMS	:	BYTE := 3;
	PUMP1_END_READ	:	BYTE := 4;
	PUMP2_STATUS	:	BYTE := 5;
	PUMP2_DATA		:	BYTE := 6;
	PUMP2_ALARMS	:	BYTE := 7;
	PUMP2_END_READ	:	BYTE := 8;
	CIR_ON_OFF1		:	BYTE := 90;
	CIR_ON_OFF2		:	BYTE := 91;
	CIR_ON_OFF_CHECK:	BYTE := 92;
	CIR_END_WRITE	:	BYTE := 93;
	ERROR_STATE		:	BYTE := 100;

END_VAR
VAR_INPUT
	ID		:	BYTE;
	Address1:	BYTE;		(* Pump 1 Modbus address *)
	Address2:	BYTE;		(* Pump 2 Modbus address *)

	(* Physical inputs (Force) *)
	CIR_RUN_REQ		: BOOL; (* External run request (no heat or cold requested) *)
	CIR_STOP_REQ	: BOOL; (* External stop request (has priority over RUN signals!) *)

	(* Physical inputs (Feedback) *)
	PumpA_AL		: BOOL; (* Alarm input signal *)
	PumpB_AL		: BOOL;
	PumpA_AUTO		: BOOL;	(* Automatic/Manual input *)
	PumpB_AUTO		: BOOL;

	(* Controls *)
	OnOff		: 	BOOL;	(* On/Off from chrono *)
	Mode		:	BYTE;	(* Working mode: 0-Both pumps works simultaneously, 1-Alternate every 24h, 2-Master/Backup *)
	InitOK		:	BOOL;

	(* Timings *)
	OnDelay		:	TIME;	(* Switch on delay *)
	OffDelay	:	TIME;	(* Switch off delay *)

	(* Modbus *)
	Refresh_Now	:	BOOL;	(* Start immediately modbus state machine *)
	retryErrMax	:	BYTE := 2;

	(* Riferimento Velocità da remoto arriva dall'esterno e mi otimizza la portata sulla mandata acqua principale *)

	VelocitaRichiesta:INT:=100;


END_VAR
VAR_IN_OUT
	ModBus		:	obj_MODBUS;
END_VAR
VAR_OUTPUT
	Ctrl_Run	:	BOOL;		(* Logical status of the device: 0: Not running (switched off), 1: running *)
	Run			:	BOOL;		(* Real status *)

	Status_Log	:	WORD;
	Status_Vis	:	DWORD;
END_VAR
VAR
	Status		:	BOOL;
	Pump_En		:	ARRAY [1..2] OF WORD;		(* Pumps enable *)

	ChangeTmr	: 	TON := (PT:=T#24h);			(* Timer that counts change time when in alternate mode *)
	ActivePump	: 	BYTE := 1;						(* Actual active pump *)
	NewActivePump	: BYTE := 1;

	(* Filters *)
	fPump_ST	: 	ARRAY [1..2] OF FLT_TAP := (INITEV:=FALSE);
	fPump_En	:	ARRAY [1..2] OF FLT_EVENT;
	fCIR_AUTO	:	ARRAY [1..2] OF FLT_TAP;
	fStatusFault:	ARRAY [1..2] OF BOOL;
	fBackup		:	FLT_EVENT := (INITEV:=FALSE);

	(* Timer manage switch on/off delay *)
	Delay		: 	TONOF;

	(* CIR data structure *)
	DataPump1	:	typ_MODBUS_CIR;
	DataPump2	:	typ_MODBUS_CIR;

	(* Modbus variables *)
	state		:	INT;
	retry		:	BYTE;
	retryErr	:	BYTE;
	ReadTmr		:	TON := (PT:=T#5s);
	fModbusAlr	: 	BOOL;

	(* Alarm and Warning counters *)
	AlarmCtr	:	BYTE;
	WarningCtr	:	BYTE;

	(* Filers on alarms and faults *)
	AlarmHw		:	ARRAY [1..2] OF FLT_TAP := (INITEV:=FALSE);
	Alarm		:	ARRAY [1..2] OF FLT_EVENT := (INITEV:=FALSE);
	Inverter	:	ARRAY [1..2] OF FLT_EVENT := (INITEV:=FALSE);
	ModbusAlr	:	FLT_EVENT := (INITEV:=FALSE);

	OldAlarmPump1	:	WORD;
	OldAlarmPump2	:	WORD;

	TimeOutModBus: TON;
	ErroreComuModBus: BOOL;

	VerificaFuctionCode: INT;
	VerificaNodoLetto: INT;

	ErroreComuModBus1: BOOL;
	ErroreComuModBus2: BOOL;
END_VAR
Init();

(* Check alarm and warning for both pumps *)
CheckFault();

PumpManager();

(* State machine to read pump parameters *)
Stm();

IF AlarmCtr>0 THEN
	Status_Log := 2;
	Status_Vis := COLOR_RED;
ELSIF WarningCtr>0 THEN
	Status_Log := 1;
	Status_Vis := COLOR_YELLOW;
ELSE
	Status_Log := 0;
	Status_Vis := COLOR_GREEN;
END_IF
END_FUNCTION_BLOCK
ACTION AddLogData:
Logger.s1:=INSERT('&CIRDM=',BYTE_TO_STRING(ID),6);
IF ID<10 THEN Logger.s1:=INSERT(Logger.s1,'0',6); END_IF

Logger.s1:=CONCAT(Logger.s1,WORD_TO_STRING(Mode));						Logger.s1:=CONCAT(Logger.s1,';');
(* PUMP 1 *)
(* NB If value equals 0x7FFF (32767) this means that it is not available -->> Change it to 0 *)
Logger.s1:=CONCAT(Logger.s1,WORD_TO_STRING(DataPump1.PumpStatus));											Logger.s1:=CONCAT(Logger.s1,';');
Logger.s1:=CONCAT(Logger.s1,INT_TO_STRING(SEL(DataPump1.PumpBoardTemp=16#7FFF,DataPump1.PumpBoardTemp,0)));	Logger.s1:=CONCAT(Logger.s1,';');
Logger.s1:=CONCAT(Logger.s1,WORD_TO_STRING(SEL(DataPump1.PumpVoltage=16#7FFF,DataPump1.PumpVoltage,0)));		Logger.s1:=CONCAT(Logger.s1,';');
Logger.s1:=CONCAT(Logger.s1,WORD_TO_STRING(SEL(DataPump1.PumpCurrent=16#7FFF,DataPump1.PumpCurrent,0)));		Logger.s1:=CONCAT(Logger.s1,';');
Logger.s1:=CONCAT(Logger.s1,WORD_TO_STRING(SEL(DataPump1.PumpPower=16#7FFF,DataPump1.PumpPower,0)));			Logger.s1:=CONCAT(Logger.s1,';');
Logger.s1:=CONCAT(Logger.s1,WORD_TO_STRING(SEL(DataPump1.PumpRPM=16#7FFF,DataPump1.PumpRPM,0)));				Logger.s1:=CONCAT(Logger.s1,';');
Logger.s1:=CONCAT(Logger.s1,WORD_TO_STRING(SEL(DataPump1.PumpHead=16#7FFF,DataPump1.PumpHead,0)));				Logger.s1:=CONCAT(Logger.s1,';');
Logger.s1:=CONCAT(Logger.s1,WORD_TO_STRING(SEL(DataPump1.PumpFlow=16#7FFF,DataPump1.PumpFlow,0)));				Logger.s1:=CONCAT(Logger.s1,';');
Logger.s1:=CONCAT(Logger.s1,WORD_TO_STRING(SEL(DataPump1.PumpLiqTemp=16#7FFF,DataPump1.PumpLiqTemp,0)));		Logger.s1:=CONCAT(Logger.s1,';');
Logger.s1:=CONCAT(Logger.s1,DWORD_TO_STRING(SEL(DataPump1.PumpOpTime=16#7FFF,DataPump1.PumpOpTime,0)));		Logger.s1:=CONCAT(Logger.s1,';');


(* PUMP 2 *)
Logger.s1:=CONCAT(Logger.s1,WORD_TO_STRING(DataPump2.PumpStatus));											Logger.s1:=CONCAT(Logger.s1,';');
Logger.s1:=CONCAT(Logger.s1,INT_TO_STRING(SEL(DataPump2.PumpBoardTemp=16#7FFF,DataPump2.PumpBoardTemp,0)));	Logger.s1:=CONCAT(Logger.s1,';');
Logger.s1:=CONCAT(Logger.s1,WORD_TO_STRING(SEL(DataPump2.PumpVoltage=16#7FFF,DataPump2.PumpVoltage,0)));		Logger.s1:=CONCAT(Logger.s1,';');
Logger.s1:=CONCAT(Logger.s1,WORD_TO_STRING(SEL(DataPump2.PumpCurrent=16#7FFF,DataPump2.PumpCurrent,0)));		Logger.s1:=CONCAT(Logger.s1,';');
Logger.s1:=CONCAT(Logger.s1,WORD_TO_STRING(SEL(DataPump2.PumpPower=16#7FFF,DataPump2.PumpPower,0)));			Logger.s1:=CONCAT(Logger.s1,';');
Logger.s1:=CONCAT(Logger.s1,WORD_TO_STRING(SEL(DataPump2.PumpRPM=16#7FFF,DataPump2.PumpRPM,0)));				Logger.s1:=CONCAT(Logger.s1,';');
Logger.s1:=CONCAT(Logger.s1,WORD_TO_STRING(SEL(DataPump2.PumpHead=16#7FFF,DataPump2.PumpHead,0)));				Logger.s1:=CONCAT(Logger.s1,';');
Logger.s1:=CONCAT(Logger.s1,WORD_TO_STRING(SEL(DataPump2.PumpFlow=16#7FFF,DataPump2.PumpFlow,0)));				Logger.s1:=CONCAT(Logger.s1,';');
Logger.s1:=CONCAT(Logger.s1,WORD_TO_STRING(SEL(DataPump2.PumpLiqTemp=16#7FFF,DataPump2.PumpLiqTemp,0)));		Logger.s1:=CONCAT(Logger.s1,';');
Logger.s1:=CONCAT(Logger.s1,DWORD_TO_STRING(SEL(DataPump2.PumpOpTime=16#7FFF,DataPump2.PumpOpTime,0)));		Logger.s1:=CONCAT(Logger.s1,';');

Logger.s1:=CONCAT(Logger.s1,WORD_TO_STRING(Status_Log));
Logger.s1:=CONCAT(Logger.s1,';');

Logger.s1:=CONCAT(Logger.s1,SEL(DataPump1.PumpFault,'0','100'));
Logger.s1:=CONCAT(Logger.s1,';');
Logger.s1:=CONCAT(Logger.s1,SEL(DataPump2.PumpFault,'0','100'));
Logger.s1:=CONCAT(Logger.s1,';');
Logger.s1:=CONCAT(Logger.s1,SEL(CIR_RUN_REQ,'0','100'));
Logger.s1:=CONCAT(Logger.s1,';');
Logger.s1:=CONCAT(Logger.s1,SEL(CIR_STOP_REQ,'0','100'));



ADDSTRING(ADR(Logger.TData), ADR(Logger.s1), Logger.TLen);
END_ACTION
ACTION CheckFault:
(*** WARNINGS ***)




(*** ALARMS ***)

(**** PUMP 1 ****)

(* Hardware alarm (physical input *)
AlarmHw[1](IN:=PumpA_AL);

IF AlarmHw[1].EVH THEN
	LogEv(EL_Alarm,EO_CIRDM,ID,3,'Scatto_Termico_A');
	AlarmCtr := AlarmCtr + 1;
END_IF

IF AlarmHw[1].EVL THEN
	LogEv(EL_Log,EO_CIRDM,ID,4,'Termico_Riarmato_A');
	AlarmCtr := SEL(AlarmCtr=0, AlarmCtr-1, 0);
END_IF

(*
(* General alarm (read by Modbus) *)
Alarm[1](IN:=(DataPump1.PumpAlarm[0] <> OldAlarmPump1));

IF Alarm[1].EVH THEN
	IF DataPump1.PumpAlarm[1] = 0 THEN
		LogEv(EL_Alarm,EO_CIRDM,ID,11,'1');
		AlarmCtr := SEL(AlarmCtr=0, AlarmCtr-1, 0);
	ELSE
		LogEv(EL_Alarm,EO_CIRDM,ID,12,WORD_TO_STRING(DataPump1.PumpAlarm[1]));
		AlarmCtr := AlarmCtr + 1;
	END_IF

	OldAlarmPump1 := DataPump1.PumpAlarm[1];
END_IF

(* Inverter pump error *)
Inverter[1](IN:=DataPump1.PumpFault);

IF Inverter[1].EVH THEN
	LogEv(EL_Alarm,EO_CIRDM,ID,9,'1');
	AlarmCtr := AlarmCtr + 1;
END_IF

IF Inverter[1].EVL THEN
	LogEv(EL_Alarm,EO_CIRDM,ID,10,'1');
	AlarmCtr := SEL(AlarmCtr=0, AlarmCtr-1, 0);
END_IF
*)

(**** PUMP 2 ****)

(* Hardware alarm (physical input *)
AlarmHw[2](IN:=PumpB_AL);

IF AlarmHw[2].EVH THEN
	LogEv(EL_Alarm,EO_CIRDM,ID,3,'Scatto_Termico_B');
	AlarmCtr := AlarmCtr + 1;
END_IF

IF AlarmHw[2].EVL THEN
	LogEv(EL_Log,EO_CIRDM,ID,4,'Termico_Riarmato_B');
	AlarmCtr := SEL(AlarmCtr=0, AlarmCtr-1, 0);
END_IF

(*
(* General alarm (read by Modbus) *)
Alarm[2](IN:=(DataPump2.PumpAlarm[0] <> OldAlarmPump2));

IF Alarm[2].EVH THEN
	IF DataPump2.PumpAlarm[0] = 0 THEN
		LogEv(EL_Log,EO_CIRDM,ID,11,'2');
		AlarmCtr := SEL(AlarmCtr=0, AlarmCtr-1, 0);
	ELSE
		LogEv(EL_Alarm,EO_CIRDM,ID,12,WORD_TO_STRING(DataPump2.PumpAlarm[0]));
		AlarmCtr := AlarmCtr + 1;
	END_IF

	OldAlarmPump2 := DataPump2.PumpAlarm[0];
END_IF

(* Inverter pump error *)
Inverter[2](IN:=DataPump2.PumpFault);

IF Inverter[2].EVH THEN
	LogEv(EL_Alarm,EO_CIRDM,ID,9,'2');
	AlarmCtr := AlarmCtr + 1;
END_IF

IF Inverter[2].EVL THEN
	LogEv(EL_Log,EO_CIRDM,ID,10,'2');
	AlarmCtr := SEL(AlarmCtr=0, AlarmCtr-1, 0);
END_IF
*)


(* Verify ModBus error	*)

ModbusAlr(IN:=FALSE );

IF ModbusAlr.EVH THEN
	LogEv(EL_Alarm,EO_CIRDM,Modbus.MB_Query.SlaveAddress,13,CONCAT('ErroreModbus',INT_TO_STRING(ModBus.MB_MASTER.MB_Error)));
END_IF

IF ModbusAlr.EVL THEN
	LogEv(EL_Log,EO_CIRDM,Modbus.MB_Query.SlaveAddress,14,'ComunicazioneModBus_OK');
END_IF
END_ACTION
ACTION Init:
IF NOT InitOK THEN

	Delay.PT_OF := SEL(OffDelay=T#0s, OffDelay, Plant_CirOffDelay);
	Delay.PT_ON := SEL(OnDelay=T#0s, OnDelay, Plant_CirOnDelay) + WORD_TO_TIME(1000*ID);

	ReadTmr.PT := WORD_TO_TIME(2000*ID);	(* 1s delay between reads of 2 different double CIRs *)

	Pump_En[1] := 1;
	Pump_En[2] := 1;

	Refresh_Now := TRUE;
	InitOK := TRUE;

END_IF
END_ACTION
ACTION PumpManager:
(*** Verify Status ***)
IF PumpA_AUTO THEN
	IF (Pump_En[1]=1 AND DataPump1.PumpStatus=2) OR (Pump_En[1]=0 AND DataPump1.PumpStatus=0) THEN fStatusFault[1] := TRUE;
	ELSE fStatusFault[1] := FALSE;
	END_IF
END_IF

IF PumpB_AUTO THEN
	IF (Pump_En[2]=1 AND DataPump2.PumpStatus=2) OR (Pump_En[2]=0 AND DataPump2.PumpStatus=0) THEN fStatusFault[2] := TRUE;
	ELSE fStatusFault[2] := FALSE;
	END_IF
END_IF

fPump_ST[1](IN:=fStatusFault[1]);
fPump_ST[2](IN:=fStatusFault[2]);

IF fPump_ST[1].EVH THEN
	LogEv(SEL(Pump_En[1]=1,EL_Alarm,EL_Wrn),EO_CIRDM,ID,SEL(Pump_En[1]=1,5,6),'1');
	WarningCtr := WarningCtr + 1;
END_IF

IF fPump_ST[1].EVL THEN WarningCtr := SEL(WarningCtr=0, WarningCtr-1, 0); END_IF

IF fPump_ST[2].EVH THEN
	LogEv(SEL(Pump_En[2]=1,EL_Alarm,EL_Wrn),EO_CIRDM,ID,SEL(Pump_En[2]=1,5,6),'2');
	WarningCtr := WarningCtr + 1;
END_IF

IF fPump_ST[2].EVL THEN WarningCtr := SEL(WarningCtr=0, WarningCtr-1, 0); END_IF


(* Verify if in Auto or Manual mode *)
fCIR_AUTO[1](IN:=PumpA_AUTO);
fCIR_AUTO[2](IN:=PumpB_AUTO);

(*** Pump A ***)
IF fCIR_AUTO[1].EVH THEN
	LogEv(EL_Log,EO_CIRDM,ID,8,'1');
	WarningCtr := SEL(WarningCtr=0, WarningCtr-1, 0);

	IF ActivePump=2 THEN Pump_En[1] := 1; END_IF
	Refresh_Now := TRUE;
END_IF

(* Manual -> Keep switched on *)
IF fCIR_AUTO[1].EVL THEN
	LogEv(EL_Wrn,EO_CIRDM,ID,7,'1');
	WarningCtr := WarningCtr + 1;

	(* Switch on pump A *)
	Pump_En[1] := 0;
(*	Run := TRUE;
	Ctrl_Run := TRUE;*)
	Refresh_Now := TRUE;
END_IF

(*** Pump B ***)
IF fCIR_AUTO[2].EVH THEN
	LogEv(EL_Log,EO_CIRDM,ID,8,'2');
	WarningCtr := SEL(WarningCtr=0, WarningCtr-1, 0);

	IF ActivePump=1 THEN Pump_En[2] := 1; END_IF
	Refresh_Now := TRUE;
END_IF

(* Manual -> Keep switched on *)
IF fCIR_AUTO[2].EVL THEN
	LogEv(EL_Wrn,EO_CIRDM,ID,7,'2');
	WarningCtr := WarningCtr + 1;

	(* Switch on pump B *)
	Pump_En[2] := 0;
(*	Ctrl_Run := TRUE;
	Run := TRUE;*)
	Refresh_Now := TRUE;
END_IF

IF PumpA_AUTO AND PumpB_AUTO THEN
	(* Verify if OnOff is changed *)
	Ctrl_Run := OnOff;
END_IF

(* Check switch on or switch off delay *)
Delay(IN:=Ctrl_Run);

(* If working mode is Alternate, count change time *)
IF Mode=1 THEN

	ChangeTmr(IN:=NOT ChangeTmr.Q);

	IF ChangeTmr.Q THEN

		NewActivePump := SEL(ActivePump=1,1,2);

		(* If no alarm on other pump, keep going with the switch *)
		IF NOT AlarmHw[NewActivePump].OUT THEN ActivePump := NewActivePump;
		ELSE LogEv(EL_Wrn,EO_CIRDM,ID,15,'');		(* Pump not switched because of other pump's failure *)
		END_IF

		(* Switch off old active pump *)
		IF ActivePump=1 THEN Pump_En[2] := 1;
		ELSE Pump_En[1] := 1;
		END_IF

		(* Write new parameters (also if not changed) *)
		Refresh_Now := TRUE;
		ChangeTmr.PT:=T#24h;
	END_IF
END_IF


(* Set output according to actual function mode *)
CASE Mode OF

	0:	(*** Simultaneous pumps working ***)
		IF PumpA_AUTO THEN

			IF CIR_STOP_REQ THEN Pump_En[1] := 1;
			ELSIF CIR_RUN_REQ THEN Pump_En[1] := 0;
			ELSE Pump_En[1] := BOOL_TO_WORD(NOT Delay.OUT);
			END_IF

			(* Set RUN signal (for external objects) *)
			IF AlarmCtr>0 THEN (*OR fPump_ST[1].OUT OR fPump_ST[2].OUT THEN*)
				Run:=FALSE;
			ELSE
				Run:=SEL(Pump_En[1]=1,TRUE,FALSE);
			END_IF
		END_IF

		IF PumpB_AUTO THEN

